// TIA Portal V17 export
// export: Created 2025-06-20T10:25:51.5107314Z, ExportSetting WithDefaults, DisplayName Totally Integrated Automation Portal, DisplayVersion V17 Update 8, DisplayName TIA Portal Openness, DisplayVersion V17 Update 8, DisplayName TIA Portal Version Control Interface, DisplayVersion V17, DisplayName SINAMICS Startdrive Advanced, DisplayVersion V17 SP2, DisplayName SINAMICS Startdrive G110M, G120, G120C, G120D, G120P, G115D, DisplayVersion V17 SP2, DisplayName SINAMICS Startdrive G130, G150, S120, S150, SINAMICS MV, S210, DisplayVersion V17 SP2, DisplayName STEP 7 Professional, DisplayVersion V17 Update 8, DisplayName SINUMERIK ONE STEP 7 Toolbox, DisplayVersion V17 Update 12, DisplayName SINUMERIK ONE PLC Basic Program Plus, DisplayVersion V17 Update 12, DisplayName SINUMERIK 840D sl STEP 7 Toolbox, DisplayVersion V17 Update 12, DisplayName STEP 7 Safety, DisplayVersion V17 Update 6, DisplayName WinCC Advanced, DisplayVersion V17 Update 8
DATA_BLOCK "DB450_ALARMS_WARNINGS_OPC_UA"   // DB450
{ S7_Optimized_Access := 'FALSE' }
VERSION : 0.1
// stored: AutoNumber false, DBAccessibleFromOPCUA true, DBAccessibleFromWebserver true, IsOnlyStoredInLoadMemory false, IsWriteProtectedInAS false
   VAR RETAIN
      ALARMS : Struct   // ALARMS MAIN NODE
         GENERAL : Struct   // GENERAL ALARMS
            "700008" : Bool;   // (RHP_SEOC) C11 Nreal<Nref
            "700009" : Bool;   // (RHP_SEOC) C11 ROTATION CONTROL FAULT
            "700010" : Bool;   // (RHP_SEOC) C11 COOLING SYSTEM OFF
            "700011" : Bool;   // (RHP_SEOC) C11 MQL OR COOLANT SYSTEM OFF
            "700012" : Bool;   // (SEOC) C11 HIGH TEMPERATURE ALARM
            "700013" : Bool;   // (SEOC) C11 PTC SENSOR HIGH TEMPERATURE ALARM
            "700014" : Bool;   // (SEOC) C11 VPM NOT READY ALARM
            "700016" : Bool;   // (RHP_SEOC) C12 Nreal<Nref
            "700017" : Bool;   // (RHP_SEOC) C12 ROTATION CONTROL FAULT
            "700018" : Bool;   // (RHP_SEOC) C12 COOLING SYSTEM OFF
            "700019" : Bool;   // (RHP_SEOC) C12 MQL OR COOLANT SYSTEM OFF
            "700020" : Bool;   // (SEOC) C12 HIGH TEMPERATURE ALARM
            "700021" : Bool;   // (SEOC) C12 PTC SENSOR HIGH TEMPERATURE ALARM
            "700022" : Bool;   // (SEOC) C12 VPM NOT READY ALARM
            "700024" : Bool;   // (RHP_SEOC) C13 Nreal<Nref
            "700025" : Bool;   // (RHP_SEOC) C13 ROTATION CONTROL FAULT
            "700026" : Bool;   // (RHP_SEOC) C13 COOLING SYSTEM OFF
            "700027" : Bool;   // (RHP_SEOC) C13 MQL OR COOLANT SYSTEM OFF
            "700028" : Bool;   // (SEOC) C13 HIGH TEMPERATURE ALARM
            "700029" : Bool;   // (SEOC) C13 PTC SENSOR HIGH TEMPERATURE ALARM
            "700030" : Bool;   // (SEOC) C13 VPM NOT READY ALARM
            "700032" : Bool;   // (RHP_SEOC) C14 Nreal<Nref
            "700033" : Bool;   // (RHP_SEOC) C14 ROTATION CONTROL FAULT
            "700034" : Bool;   // (RHP_SEOC) C14 COOLING SYSTEM OFF
            "700035" : Bool;   // (RHP_SEOC) C14 MQL OR COOLANT SYSTEM OFF
            "700036" : Bool;   // (SEOC) C14 HIGH TEMPERATURE ALARM
            "700037" : Bool;   // (SEOC) C14 PTC SENSOR HIGH TEMPERATURE ALARM
            "700038" : Bool;   // (SEOC) C14 VPM NOT READY ALARM
            "700056" : Bool;   // (RHP_SEOC) C21 Nreal<Nref
            "700057" : Bool;   // (RHP_SEOC) C21 ROTATION CONTROL FAULT
            "700058" : Bool;   // (RHP_SEOC) C21 COOLING SYSTEM OFF
            "700059" : Bool;   // (RHP_SEOC) C21 MQL OR COOLANT SYSTEM OFF
            "700060" : Bool;   // (SEOC) C21 HIGH TEMPERATURE ALARM
            "700061" : Bool;   // (SEOC) C21 PTC SENSOR HIGH TEMPERATURE ALARM
            "700062" : Bool;   // (SEOC) C21 VPM NOT READY ALARM
            "700072" : Bool;   // (RHP_SEOC) C23 Nreal<Nref
            "700073" : Bool;   // (RHP_SEOC) C23 ROTATION CONTROL FAULT
            "700074" : Bool;   // (RHP_SEOC) C23 COOLING SYSTEM OFF
            "700075" : Bool;   // (RHP_SEOC) C23 MQL OR COOLANT SYSTEM OFF
            "700076" : Bool;   // (SEOC) C23 HIGH TEMPERATURE ALARM
            "700077" : Bool;   // (SEOC) C23 PTC SENSOR HIGH TEMPERATURE ALARM
            "700078" : Bool;   // (SEOC) C23 VPM NOT READY ALARM
            "700080" : Bool;   // (RHP_SEOC) C24 Nreal<Nref
            "700081" : Bool;   // (RHP_SEOC) C24 ROTATION CONTROL FAULT
            "700082" : Bool;   // (RHP_SEOC) C24 COOLING SYSTEM OFF
            "700083" : Bool;   // (RHP_SEOC) C24 MQL OR COOLANT SYSTEM OFF
            "700084" : Bool;   // (SEOC) C24 HIGH TEMPERATURE ALARM
            "700085" : Bool;   // (SEOC) C24 PTC SENSOR HIGH TEMPERATURE ALARM
            "700086" : Bool;   // (SEOC) C24 VPM NOT READY ALARM
            "700104" : Bool;   // (IS_SEOC) AXIS E10 NOT REFERENCED
            "700111" : Bool;   // (IS_SEOC) AXIS X13 NOT REFERENCED
            "700113" : Bool;   // (IS_SEOC) AXIS Z13 NOT REFERENCED
            "700115" : Bool;   // (IS_SEOC) AXIS W11 NOT REFERENCED
            "700117" : Bool;   // (IS_SEOC) AXIS E20 NOT REFERENCED
            "700120" : Bool;   // (IS_SEOC) AXIS C22 NOT REFERENCED
            "700124" : Bool;   // (IS_SEOC) AXIS X23 NOT REFERENCED
            "700126" : Bool;   // (IS_SEOC) AXIS Z23 NOT REFERENCED
            "700128" : Bool;   // (IS_SEOC) AXIS W21 NOT REFERENCED
            "700133" : Bool;   // (IS_SEOC) AXIS C31 NOT REFERENCED
            "700400" : Bool;   // (IS) CHANNEL 1 NOT IN SOFT MODE. CHECK 20150[20]=2
            "700401" : Bool;   // (IS) PROGRAM SELECTION FAULT CHANNEL 1
            "700402" : Bool;   // (IS_SEOC) CHANNEL 1 READ AXES POSITION ALARM
            "700416" : Bool;   // (IS) CHANNEL 2 NOT IN SOFT MODE. CHECK 20150[20]=2
            "700417" : Bool;   // (IS) PROGRAM SELECTION FAULT CHANNEL 2
            "700418" : Bool;   // (IS_SEOC) CHANNEL 2 READ AXES POSITION ALARM
            "700432" : Bool;   // (IS) CHANNEL 3 NOT IN SOFT MODE. CHECK 20150[20]=2
            "700433" : Bool;   // (IS) PROGRAM SELECTION FAULT CHANNEL 3
            "700434" : Bool;   // (IS_SEOC) CHANNEL 3 READ AXES POSITION ALARM
            "700448" : Bool;   // (IS) CHANNEL 4 NOT IN SOFT MODE. CHECK 20150[20]=2
            "700449" : Bool;   // (IS) PROGRAM SELECTION FAULT CHANNEL 4
            "700450" : Bool;   // (IS_SEOC) CHANNEL 4 READ AXES POSITION ALARM
            "700464" : Bool;   // (IS) CHANNEL 5 NOT IN SOFT MODE. CHECK 20150[20]=2
            "700465" : Bool;   // (IS) PROGRAM SELECTION FAULT CHANNEL 5
            "700466" : Bool;   // (IS_SEOC) CHANNEL 5 READ AXES POSITION ALARM
            "700480" : Bool;   // (IS) CHANNEL 6 NOT IN SOFT MODE. CHECK 20150[20]=2
            "700481" : Bool;   // (IS) PROGRAM SELECTION FAULT CHANNEL 6
            "700482" : Bool;   // (IS_SEOC) CHANNEL 6 READ AXES POSITION ALARM
            "700496" : Bool;   // (IS) CHANNEL 7 NOT IN SOFT MODE. CHECK 20150[20]=2
            "700497" : Bool;   // (IS) PROGRAM SELECTION FAULT CHANNEL 7
            "700498" : Bool;   // (IS_SEOC) CHANNEL 7 READ AXES POSITION ALARM
            "700512" : Bool;   // (IS) CHANNEL 8 NOT IN SOFT MODE. CHECK 20150[20]=2
            "700513" : Bool;   // (IS) PROGRAM SELECTION FAULT CHANNEL 8
            "700514" : Bool;   // (IS_SEOC) CHANNEL 8 READ AXES POSITION ALARM
            "700528" : Bool;   // (IS) CHANNEL 9 NOT IN SOFT MODE. CHECK 20150[20]=2
            "700529" : Bool;   // (IS) PROGRAM SELECTION FAULT CHANNEL 9
            "700530" : Bool;   // (IS_SEOC) CHANNEL 9 READ AXES POSITION ALARM
            "700560" : Bool;   // (IS) FEEDBACK EMERGENCY STOP ALARM
            "700561" : Bool;   // (IS) FEEDBACK SAFETY DOORS UNIT 1 ALARM
            "700562" : Bool;   // (IS) FEEDBACK POWER ENABLE ALARM
            "700563" : Bool;   // (IS) FEEDBACK MACHINE TO ROBOT CELL SAFETY DOORS ALARM
            "700567" : Bool;   // (IS) FEEDBACK MACHINE EMERGENCY STOP ALARM
            "700568" : Bool;   // (IS) FEEDBACK LASER ENABLE CONDITIONS ALARM
            "700569" : Bool;   // (IS) FEEDBACK SAFETY DOORS UNIT 2 ALARM
            "700584" : Bool;   // (IS) TEST STOP SEQUENCE TIME EXCEEDED
            "700592" : Bool;   // (IS) BRAKE TEST AXIS X13 ALARM
            "700593" : Bool;   // (IS) BRAKE TEST AXIS W11 ALARM
            "700594" : Bool;   // (IS) BRAKE TEST AXIS Z13 ALARM
            "700595" : Bool;   // (IS) BRAKE TEST AXIS X23 ALARM
            "700596" : Bool;   // (IS) BRAKE TEST AXIS W21 ALARM
            "700597" : Bool;   // (IS) BRAKE TEST AXIS Z23 ALARM
            "700598" : Bool;   // (IS) BRAKE TEST AXIS C11 ALARM
            "700599" : Bool;   // (IS) BRAKE TEST AXIS C12 ALARM
            "700600" : Bool;   // (IS) BRAKE TEST AXIS C13 ALARM
            "700601" : Bool;   // (IS) BRAKE TEST AXIS C14 ALARM
            "700602" : Bool;   // (IS) BRAKE TEST AXIS C21 ALARM
            "700603" : Bool;   // (IS) BRAKE TEST AXIS C22 ALARM
            "700604" : Bool;   // (IS) BRAKE TEST AXIS C23 ALARM
            "700605" : Bool;   // (IS) BRAKE TEST AXIS C24 ALARM
            "700606" : Bool;   // (IS) BRAKE TEST AXIS C31 ALARM
            "700624" : Bool;   // (IS) TEST STOP INTERNAL PULSES ALARM AXIS E10
            "700625" : Bool;   // (IS) TEST STOP INTERNAL PULSES ALARM AXIS -
            "700626" : Bool;   // (IS) TEST STOP INTERNAL PULSES ALARM AXIS C11
            "700627" : Bool;   // (IS) TEST STOP INTERNAL PULSES ALARM AXIS C12
            "700632" : Bool;   // (IS) TEST STOP INTERNAL PULSES ALARM AXIS C13
            "700633" : Bool;   // (IS) TEST STOP INTERNAL PULSES ALARM AXIS C14
            "700634" : Bool;   // (IS) TEST STOP INTERNAL PULSES ALARM AXIS -
            "700635" : Bool;   // (IS) TEST STOP INTERNAL PULSES ALARM AXIS X13
            "700640" : Bool;   // (IS) TEST STOP INTERNAL PULSES ALARM AXIS -
            "700641" : Bool;   // (IS) TEST STOP INTERNAL PULSES ALARM AXIS W11
            "700642" : Bool;   // (IS) TEST STOP INTERNAL PULSES ALARM AXIS -
            "700643" : Bool;   // (IS) TEST STOP INTERNAL PULSES ALARM AXIS Z13
            "700644" : Bool;   // (IS) TEST STOP INTERNAL PULSES ALARM AXIS -
            "700645" : Bool;   // (IS) TEST STOP INTERNAL PULSES ALARM AXIS -
            "700646" : Bool;   // (IS) TEST STOP INTERNAL PULSES ALARM AXIS E20
            "700647" : Bool;   // (IS) TEST STOP INTERNAL PULSES ALARM AXIS -
            "700648" : Bool;   // (IS) TEST STOP INTERNAL PULSES ALARM AXIS C21
            "700649" : Bool;   // (IS) TEST STOP INTERNAL PULSES ALARM AXIS C22
            "700650" : Bool;   // (IS) TEST STOP INTERNAL PULSES ALARM AXIS C23
            "700651" : Bool;   // (IS) TEST STOP INTERNAL PULSES ALARM AXIS C24
            "700652" : Bool;   // (IS) TEST STOP INTERNAL PULSES ALARM AXIS -
            "700653" : Bool;   // (IS) TEST STOP INTERNAL PULSES ALARM AXIS X23
            "700654" : Bool;   // (IS) TEST STOP INTERNAL PULSES ALARM AXIS -
            "700655" : Bool;   // (IS) TEST STOP INTERNAL PULSES ALARM AXIS W21
            "700656" : Bool;   // (IS) TEST STOP INTERNAL PULSES ALARM AXIS -
            "700657" : Bool;   // (IS) TEST STOP INTERNAL PULSES ALARM AXIS Z23
            "700658" : Bool;   // (IS) TEST STOP INTERNAL PULSES ALARM AXIS -
            "700659" : Bool;   // (IS) TEST STOP INTERNAL PULSES ALARM AXIS -
            "700660" : Bool;   // (IS) TEST STOP INTERNAL PULSES ALARM AXIS C31
            "700661" : Bool;   // TEST STOP INTERNAL PULSES ALARM AXIS -
            "700662" : Bool;   // TEST STOP INTERNAL PULSES ALARM AXIS -
            "700700" : Bool;   // (IS) ERROR I-DEVICE SAFE SENDDP POWDER FEEDER ALARM
            "700701" : Bool;   // (IS) ERROR I-DEVICE SAFE SENDDP ROBOT CELL ALARM
            "700710" : Bool;   // (IS) ERROR I-DEVICE SAFE RCVDP POWDER FEEDER ALARM
            "700711" : Bool;   // (IS) ERROR I-DEVICE SAFE RCVDP ROBOT CELL ALARM
            "702400" : Bool;   // (IS) MACHINING SEQUENCE TIME EXCEEDED
            "702443" : Bool;   // (IS_SEOC) UNIT 1 STATION 3 CALIBRATION TIME EXCEEDED
            "702446" : Bool;   // (IS_SEOC) UNIT 1 STATION 0 PART CHECK TIME EXCEEDED
            "702448" : Bool;   // (IS_SEOC) PART CYCLE UNIT 1 SEQUENCE TIME EXCEEDED
            "702451" : Bool;   // (IS_SEOC) UNIT 1 STATION 0 SEQUENCE TIME EXCEEDED
            "702452" : Bool;   // (IS_SEOC) UNIT 1 STATION 1 SEQUENCE TIME EXCEEDED
            "702454" : Bool;   // (IS_SEOC) UNIT 1 STATION 3 SEQUENCE TIME EXCEEDED
            "702455" : Bool;   // (IS_SEOC) UNIT 1 STATION 4 SEQUENCE TIME EXCEEDED
            "702458" : Bool;   // (IS_SEOC) CLEAN FIXTURE UNIT 1 SEQUENCE TIME EXCEEDED
            "702459" : Bool;   // (IS_SEOC) GUIDEWAY CLEAN UNIT 1 SEQUENCE TIME EXCEEDED
            "702460" : Bool;   // (IS_SEOC) NOZZLE CLEAN UNIT 1 SEQUENCE TIME EXCEEDED
            "702461" : Bool;   // (IS_SEOC) MAINTENANCE UNIT 1 SEQUENCE TIME EXCEEDED
            "702462" : Bool;   // (IS_SEOC) RETURN TO HOME POSITION UNIT 1 STATION 0 SEQUENCE TIME EXCEEDED
            "702463" : Bool;   // (IS_SEOC) RETURN TO HOME POSITION UNIT 1 STATION 1 SEQUENCE TIME EXCEEDED
            "702465" : Bool;   // (IS_SEOC) RETURN TO HOME POSITION UNIT 1 STATION 3 SEQUENCE TIME EXCEEDED
            "702466" : Bool;   // (IS_SEOC) RETURN TO HOME POSITION UNIT 1 STATION 4 SEQUENCE TIME EXCEEDED
            "702468" : Bool;   // (IS_SEOC) UNIT 1 STATION 3 CAMERA LASER CALIBRATION SEQUENCE TIME EXCEEDED
            "702469" : Bool;   // (IS_SEOC) UNIT 1 STATION 3 CAMERA NOZZLE CALIBRATION SEQUENCE TIME EXCEEDED
            "702470" : Bool;   // (IS_SEOC) UNIT 1 STATION 3 CAMERA JET CALIBRATION SEQUENCE TIME EXCEEDED
            "702471" : Bool;   // (IS_SEOC) UNIT 1 STATION 3 CAMERA CLADDING CALIBRATION SEQUENCE TIME EXCEEDED
            "702482" : Bool;   // (IS_SEOC) UNIT 2 STATION 2 CALIBRATION TIME EXCEEDED
            "702483" : Bool;   // (IS_SEOC) UNIT 2 STATION 3 CALIBRATION TIME EXCEEDED
            "702486" : Bool;   // (IS_SEOC) UNIT 2 STATION 0 PART CHECK TIME EXCEEDED
            "702488" : Bool;   // (IS_SEOC) PART CYCLE UNIT 2 SEQUENCE TIME EXCEEDED
            "702491" : Bool;   // (IS_SEOC) UNIT 2 STATION 0 SEQUENCE TIME EXCEEDED
            "702492" : Bool;   // (IS_SEOC) UNIT 2 STATION 1 SEQUENCE TIME EXCEEDED
            "702493" : Bool;   // (IS_SEOC) UNIT 2 STATION 2 SEQUENCE TIME EXCEEDED
            "702494" : Bool;   // (IS_SEOC) UNIT 2 STATION 3 SEQUENCE TIME EXCEEDED
            "702495" : Bool;   // (IS_SEOC) UNIT 2 STATION 4 SEQUENCE TIME EXCEEDED
            "702498" : Bool;   // (IS_SEOC) CLEAN FIXTURE UNIT 2 SEQUENCE TIME EXCEEDED
            "702499" : Bool;   // (IS_SEOC) GUIDEWAY CLEAN UNIT 2 SEQUENCE TIME EXCEEDED
            "702500" : Bool;   // (IS_SEOC) NOZZLE CLEAN UNIT 2 SEQUENCE TIME EXCEEDED
            "702501" : Bool;   // (IS_SEOC) MAINTENANCE UNIT 2 SEQUENCE TIME EXCEEDED
            "702502" : Bool;   // (IS_SEOC) RETURN TO HOME POSITION UNIT 2 STATION 0 SEQUENCE TIME EXCEEDED
            "702503" : Bool;   // (IS_SEOC) RETURN TO HOME POSITION UNIT 2 STATION 1 SEQUENCE TIME EXCEEDED
            "702504" : Bool;   // (IS_SEOC) RETURN TO HOME POSITION UNIT 2 STATION 2 SEQUENCE TIME EXCEEDED
            "702505" : Bool;   // (IS_SEOC) RETURN TO HOME POSITION UNIT 2 STATION 3 SEQUENCE TIME EXCEEDED
            "702506" : Bool;   // (IS_SEOC) RETURN TO HOME POSITION UNIT 2 STATION 4 SEQUENCE TIME EXCEEDED
            "702508" : Bool;   // (IS_SEOC) UNIT 2 STATION 3 CAMERA LASER CALIBRATION SEQUENCE TIME EXCEEDED
            "702509" : Bool;   // (IS_SEOC) UNIT 2 STATION 3 CAMERA NOZZLE CALIBRATION SEQUENCE TIME EXCEEDED
            "702510" : Bool;   // (IS_SEOC) UNIT 2 STATION 3 CAMERA JET CALIBRATION SEQUENCE TIME EXCEEDED
            "702511" : Bool;   // (IS_SEOC) UNIT 2 STATION 3 CAMERA CLADDING CALIBRATION SEQUENCE TIME EXCEEDED
            "702515" : Bool;   // (IS_SEOC) UNIT 03 MEASURING STATION SEQUENCE TIME EXCEEDED
            "702516" : Bool;   // (IS_SEOC) UNIT 03 MEASURING STATION CALIBRATION SEQUENCE TIME EXCEEDED
            "702518" : Bool;   // (IS_SEOC) RETURN TO HOME POSITION UNIT 03 MEASURING SEQUENCE TIME EXCEEDED
            "702640" : Bool;   // (IS) ANY AXIS OR CHANNEL BYPASSED
            "702641" : Bool;   // (IS) ANY PROGRAMMING FAULT PRESENT
            "702642" : Bool;   // (IS) CHECK NETWORK LOGIC ALARM
            "702648" : Bool;   // (IS) LINE CONTACTOR FEEDBACK 1 ALARM
            "702649" : Bool;   // (IS) LINE CONTACTOR FEEDBACK 2 ALARM
            "702656" : Bool;   // (IS) INFEED MODULE 1 NOT READY ALARM
            "702657" : Bool;   // (SEOC) INFEED MODULE 1 OVERTEMPERATURE ALARM
            "702658" : Bool;   // (IS) INFEED MODULE 2 NOT READY ALARM
            "702659" : Bool;   // (SEOC) INFEED MODULE 2 OVERTEMPERATURE ALARM
            "702660" : Bool;   // (SEOC) NCU HEAT SINK TEMPERATURE ALARM
            "702661" : Bool;   // (SEOC) NCU LOW BATTERY ALARM
            "702662" : Bool;   // (SEOC) NCU AIR TEMPERATURE ALARM
            "702663" : Bool;   // (IS) NCK ALARM
            "702672" : Bool;   // (IS) ELECTRICAL CABINET MAIN SWITCH CIRCUIT BREAKER TRIPPED
            "702673" : Bool;   // (SEOC) ELECTRICAL CABINET COOLING UNIT 1 CIRCUIT BREAKER TRIPPED
            "702674" : Bool;   // (SEOC) ELECTRICAL CABINET COOLING UNIT 2 CIRCUIT BREAKER TRIPPED
            "702675" : Bool;   // (IS) CONTROL VOLTAGE ON ALARM
            "702677" : Bool;   // (IS) ELECTRICAL CABINET SINAMICS DRIVES CIRCUIT BREAKER 24VDC TRIPPED 1
            "702678" : Bool;   // (IS) ELECTRICAL CABINET SINAMICS DRIVES CIRCUIT BREAKER 24VDC TRIPPED 2
            "702681" : Bool;   // (IS) ELECTRICAL CABINET QFC03 CIRCUIT BREAKER TRIPPED
            "702682" : Bool;   // (IS) ELECTRICAL CABINET SINAMICS CIRCUIT BREAKER TRIPPED
            "702683" : Bool;   // (IS) FEEDBACK MAIN SWITCH OFF ALARM
            "702684" : Bool;   // (IS) ELECTRICAL CABINET OVERVOLTAGE
            "702686" : Bool;   // (SEOC) ELECTRICAL CABINET OVERTEMPERATURE ALARM
            "702689" : Bool;   // (SEOC) ELECTRICAL CABINET COOLING UNIT 1 ALARM
            "702690" : Bool;   // (SEOC) ELECTRICAL CABINET COOLING UNIT 2 ALARM
            "702694" : Bool;   // (SEOC) SENTRON PAC OVERVOLTAGE
            "702695" : Bool;   // (SEOC) SENTRON PAC OVERCURRENT
            "702697" : Bool;   // (SEOC) SENTRON PAC UNDERVOLTAGE
            "702700" : Bool;   // (IS) POWER SUPPLY DEVICE 1 ALARM
            "702703" : Bool;   // (IS) POWER SUPPLY 24V DEVICE 1 NOT OK ALARM
            "702704" : Bool;   // (IS) POWER SUPPLY 24V DEVICE 2 NOT OK ALARM
            "702705" : Bool;   // (IS) POWER SUPPLY 24V DEVICE 3 NOT OK ALARM
            "702706" : Bool;   // (IS) POWER SUPPLY 24V DEVICE 4 NOT OK ALARM
            "702707" : Bool;   // (IS) POWER SUPPLY 24V DEVICE 5 NOT OK ALARM
            "702708" : Bool;   // (IS) POWER SUPPLY 24V DEVICE 6 NOT OK ALARM
            "702709" : Bool;   // (IS) PILZ EMERGENCY STOP OK ALARM
            "702710" : Bool;   // (SEOC) SITOP BATTERY NOT OK ALARM
            "702711" : Bool;   // (SEOC) SITOP BATTERY ALARM
            "702714" : Bool;   // (IS) ETHERNET SWITCH 1 ALARM
            "702715" : Bool;   // (IS) ETHERNET SWITCH 2 ALARM
            "702716" : Bool;   // (IS) ETHERNET SWITCH 3 ALARM
            "702717" : Bool;   // (IS) ETHERNET SWITCH 4 ALARM
            "702718" : Bool;   // (IS) PROFINET CONTROL UNIT FAULT ALARM
            "702720" : Bool;   // (IS) ELECTRONIC CIRCUIT BREAKER 1 TRIPPED
            "702721" : Bool;   // (IS) ELECTRONIC CIRCUIT BREAKER 2 TRIPPED
            "702722" : Bool;   // (IS) ELECTRONIC CIRCUIT BREAKER 3 TRIPPED
            "702723" : Bool;   // (IS) ELECTRONIC CIRCUIT BREAKER 4 TRIPPED
            "702726" : Bool;   // (IS) FC40 CIRCUIT BREAKER TRIPPED
            "702727" : Bool;   // (IS) QB02 CIRCUIT BREAKER TRIPPED
            "702776" : Bool;   // (IS) SINAMICS CIRCUIT BREAKER TRIPPED ALARM
            "702777" : Bool;   // (IS) LASER UNIT 1 CIRCUIT BREAKER TRIPPED ALARM
            "702778" : Bool;   // (IS) LASER UNIT 2 CIRCUIT BREAKER TRIPPED ALARM
            "702779" : Bool;   // (IS) OERLIKON UNIT 1 CIRCUIT BREAKER TRIPPED ALARM
            "702780" : Bool;   // (IS) OERLIKON UNIT 2 CIRCUIT BREAKER TRIPPED ALARM
            "702781" : Bool;   // (IS) HEATER CIRCUIT BREAKER TRIPPED ALARM
            "702782" : Bool;   // (IS) CAMERAS CIRCUIT BREAKER 1 TRIPPED ALARM
            "702784" : Bool;   // (IS) STIRRER CIRCUIT BREAKER TRIPPED ALARM
            "702785" : Bool;   // (IS) COOLING CIRCUIT BREAKER TRIPPED ALARM
            "702786" : Bool;   // (IS) HOPPERS CIRCUIT BREAKER TRIPPED ALARM
            "702789" : Bool;   // (IS) ROBOT CELL COOLING CIRCUIT BREAKER TRIPPED ALARM
            "702790" : Bool;   // (SEOC) CIRCUIT BREAKER TRIPPED LIGHT STATION 3 ALARM
            "702793" : Bool;   // (IS) LASER UNIT 1 OK ALARM
            "702794" : Bool;   // (IS) LASER UNIT 2 OK ALARM
            "702795" : Bool;   // (SEOC) ROBOT CELL BREAKER ALARM
            "702800" : Bool;   // (IS) MAIN OPERATOR PANEL EMERGENCY STOP ACTIVE
            "702806" : Bool;   // (IS) HT10 EMERGENCY STOP ACTIVE
            "702809" : Bool;   // (IS) EMERGENCY STOP ACTIVE
            "702812" : Bool;   // (IS) ROBOT CELL EMERGENCY STOP ACTIVE
            "702814" : Bool;   // (IS) HT10 NOT READY ALARM
            "702815" : Bool;   // (IS) HT10 ERROR STATE ALARM
            "702820" : Bool;   // (SEOC) SAFETY BYPASS KEY ALARM
            "702880" : Bool;   // (IS) PROFINET NETWORK ALARM
            "702881" : Bool;   // (SEOC) PROFINET NETWORK ALARM
            "702882" : Bool;   // (RHP_SEOC) PROFINET NETWORK ALARM
            "704000" : Bool;   // (IS) UNIT 1 MAIN SAFETY DOOR NOT CLOSED AND LOCKED
            "704001" : Bool;   // (IS) UNIT 1 MAIN SAFETY DOOR NOT POSSIBLE TO UNLOCK DEPRESSURIZE PNEUMATIC DRIVE
            "704002" : Bool;   // (IS) UNIT 1 MAIN SAFETY DOOR NOT OPEN ALARM
            "704003" : Bool;   // (IS) UNIT 1 STATION 02 UNIT SAFETY DOOR NOT CLOSED AND LOCKED
            "704004" : Bool;   // (IS) UNIT 1 STATION 02 UNIT SAFETY DOOR NOT POSSIBLE TO UNLOCK DEPRESSURIZE PNEUMATIC DRIVE
            "704005" : Bool;   // (IS) UNIT 1 STATION 02 SAFETY DOOR NOT OPEN ALARM
            "704006" : Bool;   // (IS) UNIT 1 STATION 04 SAFETY DOOR NOT CLOSED AND LOCKED
            "704007" : Bool;   // (IS) UNIT 1 STATION 04 SAFETY DOOR NOT POSSIBLE TO UNLOCK DEPRESSURIZE PNEUMATIC DRIVE
            "704008" : Bool;   // (IS) UNIT 1 STATION 04 SAFETY DOOR NOT OPEN ALARM
            "704009" : Bool;   // (IS) UNIT 2 MAIN SAFETY DOOR NOT CLOSED AND LOCKED
            "704010" : Bool;   // (IS) UNIT 2 MAIN SAFETY DOOR NOT POSSIBLE TO UNLOCK DEPRESSURIZE PNEUMATIC DRIVE
            "704011" : Bool;   // (IS) UNIT 2 MAIN SAFETY DOOR NOT OPEN ALARM
            "704012" : Bool;   // (IS) UNIT 2 STATION 02 SAFETY DOOR NOT CLOSED AND LOCKED
            "704013" : Bool;   // (IS) UNIT 2 STATION 02 SAFETY DOOR NOT POSSIBLE TO UNLOCK DEPRESSURIZE PNEUMATIC DRIVE
            "704014" : Bool;   // (IS) UNIT 2 STATION 02 SAFETY DOOR NOT OPEN ALARM
            "704015" : Bool;   // (IS) UNIT 2 STATION 04 SAFETY DOOR NOT CLOSED AND LOCKED
            "704016" : Bool;   // (IS) UNIT 2 STATION 04 SAFETY DOOR NOT POSSIBLE TO UNLOCK DEPRESSURIZE PNEUMATIC DRIVE
            "704017" : Bool;   // (IS) UNIT 2 STATION 04 SAFETY DOOR NOT OPEN ALARM
            "704240" : Bool;   // (IS_SEOC) MACHINE-ROBOT CELL PART TYPE DISCORDANCY
            "704241" : Bool;   // (IS) NO PART TYPE SELECTED
            "704242" : Bool;   // (IS) MACHINE RECIPES SEQUENCE TIME EXCEEDED ALARM
            "704243" : Bool;   // (SEOC) TEST 24 HOURS DONE
            "704264" : Bool;   // (IS) ALL FIXTURES SOFTWARE DISABLED
            "704265" : Bool;   // (IS_SEOC) ALL FIXTURES UNIT 1 DISABLED
            "704266" : Bool;   // (IS_SEOC) ALL FIXTURES UNIT 2 DISABLED
            "704275" : Bool;   // (IS) UNIT 1 FIXTURE 1&4 DISABLED SOFTWARE/HARDWARE PART PRESENT ALARM
            "704276" : Bool;   // (IS) UNIT 1 FIXTURE 2&3 DISABLED SOFTWARE/HARDWARE PART PRESENT ALARM
            "704277" : Bool;   // (IS) UNIT 2 FIXTURE 1&4 DISABLED SOFTWARE/HARDWARE PART PRESENT ALARM
            "704278" : Bool;   // (IS) UNIT 2 FIXTURE 2&3 DISABLED SOFTWARE/HARDWARE PART PRESENT ALARM
            "704400" : Bool;   // (IS) ROBOT CELL INTERLOCK LIFE BIT ALARM
            "704401" : Bool;   // (IS) PRODUCTION DISCORDANCY, ALL MACHINE FIXTURES ENABLED AND ROBOT CELL COOLING DEGRADED CYCLE ACTIVE (MORE THAN 1 COOLING DISABLED)
            "704402" : Bool;   // (IS_SEOC) ROBOT FAULT ALARM UNIT 1
            "704403" : Bool;   // (IS_SEOC) ROBOT FAULT ALARM UNIT 2
            "704404" : Bool;   // (IS_SEOC) MEASURING STATION FAULT FROM CELL
            "704410" : Bool;   // (IS) POWDER INTERLOCK LIFE BIT ALARM
            "704800" : Bool;   // (RHP_SEOC) PART REJECTED AFTER INSPECTION ON DEMAND
            "704808" : Bool;   // (SEOC) PART REJECTED AFTER INSPECTION ON DEMAND
            "704832" : Bool;   // (RHP_SEOC) QUALITY PART REJECTED AFTER PART COUNT REACHED
            "704840" : Bool;   // (SEOC) QUALITY PART REJECTED AFTER PART COUNT REACHED
            "704864" : Bool;   // (RHP_SEOC) PART REJECTED AFTER PART TYPE CHANGE
            "704872" : Bool;   // (SEOC) PART REJECTED AFTER PART TYPE CHANGE
            "704896" : Bool;   // (RHP_SEOC) PART REJECTED AFTER FIRST CYCLE
            "704904" : Bool;   // (SEOC) PART REJECTED AFTER FIRST CYCLE
         END_STRUCT;
         SERVICES : Struct   // SERVICES ALARMS
            "708080" : Bool;   // (IS) PNEUMATIC BRANCH P1 PRESSURE NOT REACHED ALARM
            "708081" : Bool;   // (IS) PNEUMATIC BRANCH P1 PRESSURE SWITCH ALARM
            "708082" : Bool;   // (IS) PNEUMATIC BRANCH P1 PRESSURE MISSING ALARM
            "708083" : Bool;   // (IS) PNEUMATIC CONNECTION SENSOR 1 ALARM
            "708084" : Bool;   // (IS) PNEUMATIC CONNECTION SENSOR 2 ALARM
            "708085" : Bool;   // (SEOC) PNEUMATIC DRIVE UNBLOCK PRESSURE ALARM
            "708086" : Bool;   // (SEOC) PNEUMATIC DRIVE PRESSURE UNBLOCK SWITCH ALARM
            "708087" : Bool;   // (SEOC) PNEUMATIC PRESSURIZATION ALARM
            "708088" : Bool;   // (SEOC) PNEUMATIC PRESSURIZATION SWITCH ALARM
            "708089" : Bool;   // (SEOC) PNEUMATIC UNIT 1 GRIPPER AIR PRESSURE ALARM
            "708090" : Bool;   // (SEOC) PNEUMATIC UNIT 1 GRIPPER AIR PRESSURE SWITCH ALARM
            "708091" : Bool;   // (SEOC) PNEUMATIC UNIT 1 LABERINT PRESSURE ALARM
            "708092" : Bool;   // (SEOC) PNEUMATIC UNIT 1 LABERINT PRESSURE SWITCH ALARM
            "708093" : Bool;   // (SEOC) PNEUMATIC UNIT 1 UPPER TABLE PRESSURE ALARM
            "708094" : Bool;   // (SEOC) PNEUMATIC UNIT 1 UPPER TABLE PRESSURE SWITCH ALARM
            "708095" : Bool;   // (SEOC) PNEUMATIC UNIT 1 LOWER TABLE PRESSURE ALARM
            "708096" : Bool;   // (SEOC) PNEUMATIC UNIT 1 LOWER TABLE PRESSURE SWITCH ALARM
            "708097" : Bool;   // (SEOC) PNEUMATIC UNIT 1 CART AXIS X PRESSURE ALARM
            "708098" : Bool;   // (SEOC) PNEUMATIC UNIT 1 CART AXIS X PRESSURE SWITCH ALARM
            "708099" : Bool;   // (SEOC) PNEUMATIC UNIT 1 STATION 3 MEASUREMENT UNIT PRESSURE ALARM
            "708100" : Bool;   // (SEOC) PNEUMATIC UNIT 1 STATION 3 MEASUREMENT UNIT PRESSURE SWITCH ALARM
            "708108" : Bool;   // (IS) PNEUMATIC INPUT FLOW ALARM
            "708109" : Bool;   // (IS) PNEUMATIC INPUT TEMPERATURE ALARM
            "708112" : Bool;   // (SEOC) PNEUMATIC UNIT 2 GRIPPER AIR PRESSURE ALARM
            "708113" : Bool;   // (SEOC) PNEUMATIC UNIT 2 GRIPPER AIR PRESSURE SWITCH ALARM
            "708114" : Bool;   // (SEOC) PNEUMATIC UNIT 2 LABERINT PRESSURE ALARM
            "708115" : Bool;   // (SEOC) PNEUMATIC UNIT 2 LABERINT PRESSURE SWITCH ALARM
            "708116" : Bool;   // (SEOC) PNEUMATIC UNIT 2 UPPER TABLE PRESSURE ALARM
            "708117" : Bool;   // (SEOC) PNEUMATIC UNIT 2 UPPER TABLE PRESSURE SWITCH ALARM
            "708118" : Bool;   // (SEOC) PNEUMATIC UNIT 2 LOWER TABLE PRESSURE ALARM
            "708119" : Bool;   // (SEOC) PNEUMATIC UNIT 2 LOWER TABLE PRESSURE SWITCH ALARM
            "708120" : Bool;   // (SEOC) PNEUMATIC UNIT 2 CART AXIS X PRESSURE ALARM
            "708121" : Bool;   // (SEOC) PNEUMATIC UNIT 2 CART AXIS X PRESSURE SWITCH ALARM
            "708122" : Bool;   // (SEOC) PNEUMATIC UNIT 2 STATION 3 MEASUREMENT UNIT PRESSURE ALARM
            "708123" : Bool;   // (SEOC) PNEUMATIC UNIT 2 STATION 3 MEASUREMENT UNIT PRESSURE SWITCH ALARM
            "708160" : Bool;   // (IS) GENERAL GAS SYSTEM PRESSURE ALARM
            "708400" : Bool;   // (IS_SEOC) MACHINE COOLING SYSTEM INPUT SENSOR FLOW LOW ALARM
            "708401" : Bool;   // (IS_SEOC) MACHINE COOLING SYSTEM INPUT SENSOR FLOW HIGH ALARM
            "708402" : Bool;   // (IS_SEOC) MACHINE COOLING SYSTEM INPUT SENSOR FLOW SETPOINT ALARM
            "708403" : Bool;   // (IS_SEOC) MACHINE COOLING SYSTEM INPUT SENSOR TEMPERATURE LOW ALARM
            "708404" : Bool;   // (IS_SEOC) MACHINE COOLING SYSTEM INPUT SENSOR TEMPERATURE HIGH ALARM
            "708405" : Bool;   // (IS_SEOC) MACHINE COOLING SYSTEM INPUT SENSOR TEMPERATURE SETPOINT ALARM
            "708407" : Bool;   // (IS_SEOC) MACHINE COOLING SYSTEM OUTPUT SENSOR FLOW LOW ALARM
            "708408" : Bool;   // (IS_SEOC) MACHINE COOLING SYSTEM OUTPUT SENSOR FLOW HIGH ALARM
            "708409" : Bool;   // (IS_SEOC) MACHINE COOLING SYSTEM OUTPUT SENSOR FLOW SETPOINT ALARM
            "708410" : Bool;   // (IS_SEOC) MACHINE COOLING SYSTEM OUTPUT SENSOR TEMPERATURE LOW ALARM
            "708411" : Bool;   // (IS_SEOC) MACHINE COOLING SYSTEM OUTPUT SENSOR TEMPERATURE HIGH ALARM
            "708412" : Bool;   // (IS_SEOC) MACHINE COOLING SYSTEM OUTPUT SENSOR TEMPERATURE SETPOINT ALARM
            "708417" : Bool;   // (SEOC) SHIELD AUXILIARY COOLING SYSTEM BREAKER TRIPPED ALARM
            "708418" : Bool;   // (SEOC) SHIELD AUXILIARY COOLING SYSTEM CONTACTOR FEEDBACK ALARM
            "708419" : Bool;   // (SEOC) SHIELD AUXILIARY COOLING SYSTEM LOW LEVEL ALARM
            "708420" : Bool;   // (SEOC) SHIELD AUXILIARY COOLING SYSTEM OVERTEMPERATURE ALARM
            "708423" : Bool;   // (SEOC) U01 SHIELD AUXILIARY COOLING SYSTEM FLOW FEEDBACK ALARM
            "708424" : Bool;   // (SEOC) U01 SHIELD AUXILIARY COOLING SYSTEM FLOW LOW ALARM
            "708425" : Bool;   // (SEOC) U01 SHIELD AUXILIARY COOLING SYSTEM FLOW HIGH ALARM
            "708426" : Bool;   // (SEOC) U01 SHIELD AUXILIARY COOLING SYSTEM TEMPERATURE LOW ALARM
            "708427" : Bool;   // (SEOC) U01 SHIELD AUXILIARY COOLING SYSTEM TEMPERATURE HIGH ALARM
            "708428" : Bool;   // (SEOC) U01 SHIELD AUXILIARY COOLING SYSTEM FLOW SETPOINT ALARM
            "708429" : Bool;   // (SEOC) U01 SHIELD AUXILIARY COOLING SYSTEM TEMPERATURE SETPOINT ALARM
            "708432" : Bool;   // (SEOC) U02 SHIELD AUXILIARY COOLING SYSTEM FLOW FEEDBACK ALARM
            "708433" : Bool;   // (SEOC) U02 SHIELD AUXILIARY COOLING SYSTEM FLOW LOW ALARM
            "708434" : Bool;   // (SEOC) U02 SHIELD AUXILIARY COOLING SYSTEM FLOW HIGH ALARM
            "708435" : Bool;   // (SEOC) U02 SHIELD AUXILIARY COOLING SYSTEM TEMPERATURE LOW ALARM
            "708436" : Bool;   // (SEOC) U02 SHIELD AUXILIARY COOLING SYSTEM TEMPERATURE HIGH ALARM
            "708437" : Bool;   // (SEOC) U02 SHIELD AUXILIARY COOLING SYSTEM FLOW SETPOINT ALARM
            "708438" : Bool;   // (SEOC) U02 SHIELD AUXILIARY COOLING SYTEM TEMPERATURE SETPOINT ALARM
            "708443" : Bool;   // (SEOC) COOLING BUFFER AUXILIARY COOLING SYSTEM BREAKER TRIPPED ALARM
            "708444" : Bool;   // (SEOC) COOLING BUFFER AUXILIARY COOLING SYSTEM CONTACTOR FEEDBACK ALARM
            "708445" : Bool;   // (SEOC) COOLING BUFFER AUXILIARY COOLING SYSTEM LOW LEVEL ALARM
            "708446" : Bool;   // (SEOC) COOLING BUFFER AUXILIARY COOLING SYSTEM OVERTEMPERATURE ALARM
            "708449" : Bool;   // (SEOC) U01 COOLING BUFFER AUXILIARY COOLING SYSTEM FLOW FEEDBACK ALARM
            "708450" : Bool;   // (SEOC) U01 COOLING BUFFER AUXILIARY COOLING SYSTEM FLOW LOW ALARM
            "708451" : Bool;   // (SEOC) U01 COOLING BUFFER AUXILIARY COOLING SYSTEM FLOW HIGH ALARM
            "708452" : Bool;   // (SEOC) U01 COOLING BUFFER AUXILIARY COOLING SYSTEM TEMPERATURE LOW ALARM
            "708453" : Bool;   // (SEOC) U01 COOLING BUFFER AUXILIARY COOLING SYSTEM TEMPERATURE HIGH ALARM
            "708454" : Bool;   // (SEOC) U01 COOLING BUFFER AUXILIARY COOLING SYSTEM FLOW SETPOINT ALARM
            "708455" : Bool;   // (SEOC) U01 COOLING BUFFER AUXILIARY COOLING SYSTEM TEMPERATURE SETPOINT ALARM
            "708458" : Bool;   // (SEOC) U02 COOLING BUFFER AUXILIARY COOLING SYSTEM FLOW FEEDBACK ALARM
            "708459" : Bool;   // (SEOC) U02 COOLING BUFFER AUXILIARY COOLING SYSTEM FLOW LOW ALARM
            "708460" : Bool;   // (SEOC) U02 COOLING BUFFER AUXILIARY COOLING SYSTEM FLOW HIGH ALARM
            "708461" : Bool;   // (SEOC) U02 COOLING BUFFER AUXILIARY COOLING SYSTEM TEMPERATURE LOW ALARM
            "708462" : Bool;   // (SEOC) U02 COOLING BUFFER AUXILIARY COOLING SYSTEM TEMPERATURE HIGH ALARM
            "708463" : Bool;   // (SEOC) U02 COOLING BUFFER AUXILIARY COOLING SYSTEM FLOW SETPOINT ALARM
            "708464" : Bool;   // (SEOC) U02 COOLING BUFFER AUXILIARY COOLING SYSTEM TEMPERATURE SETPOINT ALARM
            "708800" : Bool;   // (SEOC) PROGRESSIVE LUBRICATION CIRCUIT BREAKER TRIPPED
            "708801" : Bool;   // (SEOC) PROGRESSIVE LUBRICATION LOW LEVEL ALARM
            "708802" : Bool;   // (SEOC) PROGRESSIVE LUBRICATION OVERPRESSURE ALARM
            "708803" : Bool;   // (SEOC) PROGRESSIVE LUBRICATION BRANCH 1 CYCLE NOT DONE ALARM
            "708804" : Bool;   // (SEOC) PROGRESSIVE LUBRICATION BRANCH 2 CYCLE NOT DONE ALARM
            "708805" : Bool;   // (SEOC) PROGRESSIVE LUBRICATION BRANCH 3 CYCLE NOT DONE ALARM
            "708806" : Bool;   // (SEOC) PROGRESSIVE LUBRICATION BRANCH 4 CYCLE NOT DONE ALARM
            "708960" : Bool;   // (SEOC) MACHINE ASPIRATION SYSTEM ALARM
            "709040" : Bool;   // (IS_SEOC) UNIT 1 ASPIRATION SYSTEM PRESSURE TOO HIGH ALARM
            "709041" : Bool;   // (IS_SEOC) UNIT 1 ASPIRATION SYSTEM PRESSURE TOO LOW ALARM
            "709051" : Bool;   // (IS_SEOC) UNIT 1 STATION 1 ASPIRATION ACTIVATION SIMULTANEITY ALARM
            "709052" : Bool;   // (IS_SEOC) UNIT 1 STATION 1 ASPIRATION ACTIVATION TIME EXCEEDED ALARM
            "709053" : Bool;   // (IS_SEOC) UNIT 1 STATION 1 ASPIRATION ACTIVATION SWITCH ON ALARM
            "709054" : Bool;   // (IS_SEOC) UNIT 1 STATION 1 ASPIRATION ACTIVATION SWITCH OFF ALARM
            "709071" : Bool;   // (IS_SEOC) UNIT 1 STATION 3 ASPIRATION ACTIVATION SIMULTANEITY ALARM
            "709072" : Bool;   // (IS_SEOC) UNIT 1 STATION 3 ASPIRATION ACTIVATION TIME EXCEEDED ALARM
            "709073" : Bool;   // (IS_SEOC) UNIT 1 STATION 3 ASPIRATION ACTIVATION SWITCH ON ALARM
            "709074" : Bool;   // (IS_SEOC) UNIT 1 STATION 3 ASPIRATION ACTIVATION SWITCH OFF ALARM
            "709120" : Bool;   // (IS_SEOC) UNIT 2 ASPIRATION SYSTEM PRESSURE TOO HIGH ALARM
            "709121" : Bool;   // (IS_SEOC) UNIT 2 ASPIRATION SYSTEM PRESSURE TOO LOW ALARM
            "709131" : Bool;   // (IS_SEOC) UNIT 2 STATION 1 ASPIRATION ACTIVATION SIMULTANEITY ALARM
            "709132" : Bool;   // (IS_SEOC) UNIT 2 STATION 1 ASPIRATION ACTIVATION TIME EXCEEDED ALARM
            "709133" : Bool;   // (IS_SEOC) UNIT 2 STATION 1 ASPIRATION ACTIVATION SWITCH ON ALARM
            "709134" : Bool;   // (IS_SEOC) UNIT 2 STATION 1 ASPIRATION ACTIVATION SWITCH OFF ALARM
            "709151" : Bool;   // (IS_SEOC) UNIT 2 STATION 3 ASPIRATION ACTIVATION SIMULTANEITY ALARM
            "709152" : Bool;   // (IS_SEOC) UNIT 2 STATION 3 ASPIRATION ACTIVATION TIME EXCEEDED ALARM
            "709153" : Bool;   // (IS_SEOC) UNIT 2 STATION 3 ASPIRATION ACTIVATION SWITCH ON ALARM
            "709154" : Bool;   // (IS_SEOC) UNIT 2 STATION 3 ASPIRATION ACTIVATION SWITCH OFF ALARM
            "709161" : Bool;   // (IS_SEOC) UNIT 2 STATION 4 ASPIRATION ACTIVATION SIMULTANEITY ALARM
         END_STRUCT;
         UNIT_01 : Struct   // UNIT 01 ALARMS
            "716000" : Bool;   // (IS_SEOC) UNIT 1 FIXTURE 1 PART TYPE DISCORDANCY ALARM
            "716001" : Bool;   // (IS_SEOC) UNIT 1 FIXTURE 2 PART TYPE DISCORDANCY ALARM
            "716002" : Bool;   // (IS_SEOC) UNIT 1 FIXTURE 3 PART TYPE DISCORDANCY ALARM
            "716003" : Bool;   // (IS_SEOC) UNIT 1 FIXTURE 4 PART TYPE DISCORDANCY ALARM
            "716008" : Bool;   // (RHP_SEOC) UNIT 1 FIXTURE 1 PART PRESENT DISCORDANCY ALARM
            "716009" : Bool;   // (RHP_SEOC) UNIT 1 FIXTURE 2 PART PRESENT DISCORDANCY ALARM
            "716010" : Bool;   // (RHP_SEOC) UNIT 1 FIXTURE 3 PART PRESENT DISCORDANCY ALARM
            "716011" : Bool;   // (RHP_SEOC) UNIT 1 FIXTURE 4 PART PRESENT DISCORDANCY ALARM
            "716024" : Bool;   // (IS_SEOC) UNIT 1 FIXTURE 1 PART ORIENTATION DISCORDANCY ALARM
            "716025" : Bool;   // (IS_SEOC) UNIT 1 FIXTURE 2 PART ORIENTATION DISCORDANCY ALARM
            "716026" : Bool;   // (IS_SEOC) UNIT 1 FIXTURE 3 PART ORIENTATION DISCORDANCY ALARM
            "716027" : Bool;   // (IS_SEOC) UNIT 1 FIXTURE 4 PART ORIENTATION DISCORDANCY ALARM
            "716032" : Bool;   // (RHP_SEOC) UNIT 1 FIXTURE 1 NOT CLAMPED DURING MACHINING ALARM
            "716033" : Bool;   // (RHP_SEOC) UNIT 1 FIXTURE 2 NOT CLAMPED DURING MACHINING ALARM
            "716034" : Bool;   // (RHP_SEOC) UNIT 1 FIXTURE 3 NOT CLAMPED DURING MACHINING ALARM
            "716035" : Bool;   // (RHP_SEOC) UNIT 1 FIXTURE 4 NOT CLAMPED DURING MACHINING ALARM
            STATION_3_MEASURING : Struct   // STATION 3 MEASURING ALARMS
               "716480" : Bool;   // (IS_SEOC) UNIT 1 STATION 3 MEASURING LAST CALIBRATION OUT OF RANGE IN FIXTURE 1 ALARM
               "716481" : Bool;   // (IS_SEOC) UNIT 1 STATION 3 MEASURING LAST CALIBRATION OUT OF RANGE IN FIXTURE 2 ALARM
               "716482" : Bool;   // (IS_SEOC) UNIT 1 STATION 3 MEASURING LAST CALIBRATION OUT OF RANGE IN FIXTURE 3 ALARM
               "716483" : Bool;   // (IS_SEOC) UNIT 1 STATION 3 MEASURING LAST CALIBRATION OUT OF RANGE IN FIXTURE 4 ALARM
               "716488" : Bool;   // (IS_SEOC) UNIT 1 STATION 3 MEASURING COMPUTER CONNECTION CALL ERROR
               "716489" : Bool;   // (IS_SEOC) UNIT 1 STATION 3 MEASURING COMPUTER GET INDEX LIST CALL ERROR
               "716490" : Bool;   // (IS_SEOC) UNIT 1 STATION 3 MEASURING COMPUTER GET HANDLE LIST CALL ERROR
               "716491" : Bool;   // (IS_SEOC) UNIT 1 STATION 3 MEASURING COMPUTER GET METHOD LIST CALL ERROR
               "716492" : Bool;   // (IS_SEOC) UNIT 1 STATION 3 MEASURING COMPUTER RELEASE HANDLE LIST CALL ERROR
               "716493" : Bool;   // (IS_SEOC) UNIT 1 STATION 3 MEASURING COMPUTER RELEASE METHOD HANDLE LIST CALL ERROR
               "716494" : Bool;   // (IS_SEOC) UNIT 1 STATION 3 MEASURING COMPUTER DISCONNECT CALL ERROR
               "716500" : Bool;   // (IS_SEOC) UNIT 1 STATION 3 MEASURING COMPUTER ERROR: PROFILER CONFIGURATION (ISSUES WITH THE PROFILOMETER CONFIGURATION)
               "716501" : Bool;   // (IS_SEOC) UNIT 1 STATION 3 MEASURING COMPUTER ERROR: ANALYZER CONFIGURATION (ERROR OCCURRED WHILE VERIFYING THE CONFIGURATION FILES)
               "716502" : Bool;   // (IS_SEOC) UNIT 1 STATION 3 MEASURING COMPUTER ERROR: DMC STRUCTURE (PROBLEMS READING THE DMC STRING)
               "716503" : Bool;   // (IS_SEOC) UNIT 1 STATION 3 MEASURING COMPUTER ERROR: ACQUISITION (UNABLE TO ACQUIRE PROFILES FROM THE PROFILOMETER)
               "716504" : Bool;   // (IS_SEOC) UNIT 1 STATION 3 MEASURING COMPUTER ERROR: PROFILE INITIALIZATION (FAILED TO INITIALIZE THE PROFILOMETER)
               "716505" : Bool;   // (IS_SEOC) UNIT 1 STATION 3 MEASURING COMPUTER ERROR: DISTANCE CALCULATION (ISSUES EXECUTING THE DISTANCE CALCULATION ALGORITHM)
               "716506" : Bool;   // (IS_SEOC) UNIT 1 STATION 3 MEASURING COMPUTER ERROR: LAYER GROWTH ANALYSIS (ISSUES EXECUTING THE LAYER GROWTH ALGORITHM)
               "716507" : Bool;   // (IS_SEOC) UNIT 1 STATION 3 MEASURING COMPUTER ERROR: STORAGE ERROR (ERROR ATTEMPTING TO STORE DATA)
               "716508" : Bool;   // (IS_SEOC) UNIT 1 STATION 3 MEASURING COMPUTER ERROR: DATABASE CONNECTION ALARM (CALIBRATION CHECK OR MEASURE SAVE NOT POSSIBLE)
               "716509" : Bool;   // (IS_SEOC) UNIT 1 STATION 3 MEASURING COMPUTER ERROR: CALIBRATION PROCEDURE (CALIBRATION FAILED)
               "716510" : Bool;   // (IS_SEOC) UNIT 1 STATION 3 MEASURING COMPUTER ERROR: CALIBRATION MISSING IN FIXTURE 1 (CALIBRATION MISSING OR FILE NOT FOUND)
               "716511" : Bool;   // (IS_SEOC) UNIT 1 STATION 3 MEASURING COMPUTER ERROR: CALIBRATION MISSING IN FIXTURE 2 (CALIBRATION MISSING OR FILE NOT FOUND)
               "716512" : Bool;   // (IS_SEOC) UNIT 1 STATION 3 MEASURING COMPUTER ERROR: CALIBRATION MISSING IN FIXTURE 3 (CALIBRATION MISSING OR FILE NOT FOUND)
               "716513" : Bool;   // (IS_SEOC) UNIT 1 STATION 3 MEASURING COMPUTER ERROR: CALIBRATION MISSING IN FIXTURE 4 (CALIBRATION MISSING OR FILE NOT FOUND)
               "716514" : Bool;   // (IS_SEOC) UNIT 1 STATION 3 MEASURING COMPUTER ERROR: PLC-PC MAJOR VERSIONS MISMATCH
               "716515" : Bool;   // (SEOC) UNIT 1 STATION 3 MEASURING COMPUTER ERROR: INITIALIZING PROFILOMETER
               "716520" : Bool;   // (IS_SEOC) UNIT 1 STATION 3 MEASURING COMPUTER NOZZLE SURFACE DISTANCE UPDATE ALARM
               "716530" : Bool;   // (IS_SEOC) UNIT 1 STATION 3 MEASURING COMPUTER START NOOZLE MEASUREMENT METHOD CALL EXECUTION ERROR
               "716531" : Bool;   // (IS_SEOC) UNIT 1 STATION 3 MEASURING COMPUTER START NOOZLE MEASUREMENT METHOD WORKING OR BLOCKED ERROR
               "716546" : Bool;   // (IS_SEOC) UNIT 1 STATION 3 MEASURING COMPUTER START LAYER THICKNESS MEASUREMENT METHOD CALL EXECUTION ERROR
               "716547" : Bool;   // (IS_SEOC) UNIT 1 STATION 3 MEASURING COMPUTER START LAYER THICKNESS MEASUREMENT METHOD WORKING OR BLOCKED ERROR
               "716554" : Bool;   // (IS_SEOC) UNIT 1 STATION 3 MEASURING COMPUTER STOP LAYER THICKNESS MEASUREMENT METHOD CALL EXECUTION ERROR
               "716555" : Bool;   // (IS_SEOC) UNIT 1 STATION 3 MEASURING COMPUTER STOP LAYER THICKNESS MEASUREMENT METHOD WORKING OR BLOCKED ERROR
               "716562" : Bool;   // (IS_SEOC) UNIT 1 STATION 3 MEASURING COMPUTER CALIBRATING METHOD CALL EXECUTION ERROR
               "716563" : Bool;   // (IS_SEOC) UNIT 1 STATION 3 MEASURING COMPUTER CALIBRATING METHOD WORKING OR BLOCKED ERROR
               "716570" : Bool;   // (IS_SEOC) UNIT 1 STATION 3 MEASURING COMPUTER RESET METHOD CALL EXECUTION ERROR
               "716571" : Bool;   // (IS_SEOC) UNIT 1 STATION 3 MEASURING COMPUTER RESET METHOD WORKING OR BLOCKED ERROR
               "716578" : Bool;   // (IS_SEOC) UNIT 1 STATION 3 MEASURING COMPUTER READ VARIABLES METHOD CALL EXECUTION ERROR
               "716579" : Bool;   // (IS_SEOC) UNIT 1 STATION 3 MEASURING COMPUTER READ VARIABLES METHOD WORKING OR BLOCKED ERROR
            END_STRUCT;
            STATION_3_COAXIAL : Struct   // STATION 3 COAXIAL ALARMS
               "716640" : Bool;   // (IS_SEOC) UNIT 1 STATION 3 CAMERA COMPUTER ERROR: FAILED TO CONNECT TO CAMERA (UNABLE TO GET IMAGES FROM CAMERA)
               "716641" : Bool;   // (IS_SEOC) UNIT 1 STATION 3 CAMERA COMPUTER ERROR: FAILED TO SET CAMERA PARAMETERS (UNABLE TO SET CAMERA PARAMETERS (EXPOSURE-TIME & GAIN) FROM CURRENT IMAGES)
               "716642" : Bool;   // (IS_SEOC) UNIT 1 STATION 3 CAMERA COMPUTER ERROR: NEW LASER CALIBRATION REQUIRED (CURRENT CALIBRATION PARAMETERS DO NOT MEEST RECENT ANALYSIS REQUISITES)
               "716643" : Bool;   // (IS_SEOC) UNIT 1 STATION 3 CAMERA COMPUTER ERROR: NEW NOZZLE CALIBRATION REQUIRED (CURRENT CALIBRATION PARAMETERS DO NOT MEEST RECENT ANALYSIS REQUISITES)
               "716644" : Bool;   // (IS_SEOC) UNIT 1 STATION 3 CAMERA COMPUTER ERROR: NEW JET CALIBRATION REQUIRED (CURRENT CALIBRATION PARAMETERS DO NOT MEEST RECENT ANALYSIS REQUISITES)
               "716645" : Bool;   // (IS_SEOC) UNIT 1 STATION 3 CAMERA COMPUTER ERROR: NEW CLADDING CALIBRATION REQUIRED (CURRENT CALIBRATION PARAMETERS DO NOT MEEST RECENT ANALYSIS REQUISITES)
               "716646" : Bool;   // (IS_SEOC) UNIT 1 STATION 3 CAMERA COMPUTER ERROR: HIGH NUMBER OF DEAD PIXELS (THE NUMBER OF DEAD-PIXELS EXCEEDS A CONFIGURED NUMBER)
               "716647" : Bool;   // (IS_SEOC) UNIT 1 STATION 3 CAMERA COMPUTER ERROR: NO LIGHT DETECTED (NO LIGHT OR BLANK IMAGE DETECTED)
               "716648" : Bool;   // (IS_SEOC) UNIT 1 STATION 3 CAMERA COMPUTER ERROR: NO LASER DETECTED (NO LASER SPOT DETECTED)
               "716649" : Bool;   // (IS_SEOC) UNIT 1 STATION 3 CAMERA COMPUTER ERROR: NO NOZZLE DETECTED (UNABLE TO DETECT ANY CAPSULE-SHAPED NOZZLE IN THE IMAGE)
               "716651" : Bool;   // (IS_SEOC) UNIT 1 STATION 3 CAMERA COMPUTER ERROR: NO LASER PATTERN DETECTED (NO LASER PATERN HAS BEEN DETECTED IN THE IMAGE)
               "716652" : Bool;   // (IS_SEOC) UNIT 1 STATION 3 CAMERA COMPUTER ERROR: NOT ANALYZED
               "716653" : Bool;   // (IS_SEOC) UNIT 1 STATION 3 CAMERA COMPUTER ERROR: FAILED TO OBTAIN SCALE FACTOR
               "716654" : Bool;   // (IS_SEOC) UNIT 1 STATION 3 CAMERA COMPUTER ERROR: UNALIGNED POWDER FLOW VORTEX
               "716655" : Bool;   // (IS_SEOC) UNIT 1 STATION 3 CAMERA COMPUTER ERROR: JET MALFUNCTION
               "716656" : Bool;   // (IS_SEOC) UNIT 1 STATION 3 CAMERA COMPUTER ERROR: UNCALIBRATED
               "716657" : Bool;   // (IS_SEOC) UNIT 1 STATION 3 CAMERA COMPUTER ERROR: PLC-PC MAJOR VERSIONS MISMATCH
               "716658" : Bool;   // (IS_SEOC) UNIT 1 STATION 3 CAMERA COMPUTER ERROR: NO MELT POOL DETECTED
               "716659" : Bool;   // (IS_SEOC) UNIT 1 STATION 3 CAMERA COMPUTER ERROR: NO DATA BASE CONNECTION
               "716660" : Bool;   // (IS_SEOC) UNIT 1 STATION 3 CAMERA COMPUTER ERROR: NO HALO DETECTED
               "716661" : Bool;   // (IS_SEOC) UNIT 1 STATION 3 CAMERA COMPUTER ERROR: STORAGE ERROR
               "716662" : Bool;   // (SEOC) UNIT 1 STATION 3 CAMERA COMPUTER ERROR: INITIALIZING CAMERA
               "716663" : Bool;   // (IS_SEOC) UNIT 1 STATION 3 CAMERA COMPUTER ERROR: NOZZLE CONTAMINATION DETECTED
               "716664" : Bool;   // (IS_SEOC) UNIT 1 STATION 3 CAMERA COMPUTER ERROR: INVALID CONFIGURATION
               "716672" : Bool;   // (IS_SEOC) UNIT 1 STATION 3 CAMERA COMPUTER CONNECTION CALL ERROR
               "716673" : Bool;   // (IS_SEOC) UNIT 1 STATION 3 CAMERA COMPUTER GET INDEX LIST CALL ERROR
               "716674" : Bool;   // (IS_SEOC) UNIT 1 STATION 3 CAMERA COMPUTER GET HANDLE LIST CALL ERROR
               "716675" : Bool;   // (IS_SEOC) UNIT 1 STATION 3 CAMERA COMPUTER GET METHOD CALIBRATIONS LIST CALL ERROR
               "716676" : Bool;   // (IS_SEOC) UNIT 1 STATION 3 CAMERA COMPUTER GET METHOD ANALISIS LIST CALL ERROR
               "716677" : Bool;   // (IS_SEOC) UNIT 1 STATION 3 CAMERA COMPUTER RELEASE HANDLE LIST CALL ERROR
               "716678" : Bool;   // (IS_SEOC) UNIT 1 STATION 3 CAMERA COMPUTER RELEASE METHOD HANDLE LIST CALL ERROR
               "716679" : Bool;   // (IS_SEOC) UNIT 1 STATION 3 CAMERA COMPUTER DISCONNECT CALL ERROR
               "716680" : Bool;   // (IS_SEOC) UNIT 1 STATION 3 CAMERA COMPUTER DISCONNECT ALARM
               "716720" : Bool;   // (IS_SEOC) UNIT 1 STATION 3 COAXIAL CAMERA START LASER CALIBRATION METHOD CONNECTION ALARM
               "716721" : Bool;   // (IS_SEOC) UNIT 1 STATION 3 COAXIAL CAMERA START LASER CALIBRATION METHOD WORKING OR BLOCKED ALARM
               "716728" : Bool;   // (IS_SEOC) UNIT 1 STATION 3 COAXIAL CAMERA START NOZZLE CALIBRATION METHOD CONNECTION ALARM
               "716729" : Bool;   // (IS_SEOC) UNIT 1 STATION 3 COAXIAL CAMERA START NOZZLE CALIBRATION METHOD WORKING OR BLOCKED ALARM
               "716736" : Bool;   // (IS_SEOC) UNIT 1 STATION 3 COAXIAL CAMERA START JET CALIBRATION METHOD CONNECTION ALARM
               "716737" : Bool;   // (IS_SEOC) UNIT 1 STATION 3 COAXIAL CAMERA START JET CALIBRATION METHOD WORKING OR BLOCKED ALARM
               "716744" : Bool;   // (IS_SEOC) UNIT 1 STATION 3 COAXIAL CAMERA START CLADDING CALIBRATION METHOD CONNECTION ALARM
               "716745" : Bool;   // (IS_SEOC) UNIT 1 STATION 3 COAXIAL CAMERA START CLADDING CALIBRATION METHOD WORKING OR BLOCKED ALARM
               "716752" : Bool;   // (IS_SEOC) UNIT 1 STATION 3 COAXIAL CAMERA START NOZZLE ANALISIS METHOD CONNECTION ALARM
               "716753" : Bool;   // (IS_SEOC) UNIT 1 STATION 3 COAXIAL CAMERA START NOZZLE ANALISIS METHOD WORKING OR BLOCKED ALARM
               "716760" : Bool;   // (IS_SEOC) UNIT 1 STATION 3 COAXIAL CAMERA START JET ANALISIS METHOD CONNECTION ALARM
               "716761" : Bool;   // (IS_SEOC) UNIT 1 STATION 3 COAXIAL CAMERA START JET ANALISIS METHOD WORKING OR BLOCKED ALARM
               "716768" : Bool;   // (IS_SEOC) UNIT 1 STATION 3 COAXIAL CAMERA START CLADDING ANALISIS METHOD CONNECTION ALARM
               "716769" : Bool;   // (IS_SEOC) UNIT 1 STATION 3 COAXIAL CAMERA START CLADDING ANALISIS METHOD WORKING OR BLOCKED ALARM
               "716776" : Bool;   // (IS_SEOC) UNIT 1 STATION 3 COAXIAL CAMERA STOP METHODS CONNECTION ALARM
               "716777" : Bool;   // (IS_SEOC) UNIT 1 STATION 3 COAXIAL CAMERA STOP METHODS METHOD WORKING OR BLOCKED ALARM
               "716784" : Bool;   // (IS_SEOC) UNIT 1 STATION 3 COAXIAL CAMERA RESET PC METHOD CONNECTION ALARM
               "716785" : Bool;   // (IS_SEOC) UNIT 1 STATION 3 COAXIAL CAMERA RESET PC METHOD WORKING OR BLOCKED ALARM
               "716792" : Bool;   // (IS_SEOC) UNIT 1 STATION 3 COAXIAL CAMERA READ VARIABLES METHOD CONNECTION ALARM
               "716793" : Bool;   // (IS_SEOC) UNIT 1 STATION 3 COAXIAL CAMERA READ VARIABLES METHOD WORKING OR BLOCKED ALARM
            END_STRUCT;
         END_STRUCT;
         UNIT_02 : Struct   // UNIT 02 ALARMS
            "720000" : Bool;   // (IS_SEOC) UNIT 2 FIXTURE 1 PART TYPE DISCORDANCY ALARM
            "720001" : Bool;   // (IS_SEOC) UNIT 2 FIXTURE 2 PART TYPE DISCORDANCY ALARM
            "720002" : Bool;   // (IS_SEOC) UNIT 2 FIXTURE 3 PART TYPE DISCORDANCY ALARM
            "720003" : Bool;   // (IS_SEOC) UNIT 2 FIXTURE 4 PART TYPE DISCORDANCY ALARM
            "720008" : Bool;   // (RHP_SEOC) UNIT 2 FIXTURE 1 PART PRESENT DISCORDANCY ALARM
            "720009" : Bool;   // (RHP_SEOC) UNIT 2 FIXTURE 2 PART PRESENT DISCORDANCY ALARM
            "720010" : Bool;   // (RHP_SEOC) UNIT 2 FIXTURE 3 PART PRESENT DISCORDANCY ALARM
            "720011" : Bool;   // (RHP_SEOC) UNIT 2 FIXTURE 4 PART PRESENT DISCORDANCY ALARM
            "720024" : Bool;   // (IS_SEOC) UNIT 2 FIXTURE 1 PART ORIENTATION DISCORDANCY ALARM
            "720025" : Bool;   // (IS_SEOC) UNIT 2 FIXTURE 2 PART ORIENTATION DISCORDANCY ALARM
            "720026" : Bool;   // (IS_SEOC) UNIT 2 FIXTURE 3 PART ORIENTATION DISCORDANCY ALARM
            "720027" : Bool;   // (IS_SEOC) UNIT 2 FIXTURE 4 PART ORIENTATION DISCORDANCY ALARM
            "720032" : Bool;   // (RHP_SEOC) UNIT 2 FIXTURE 1 NOT CLAMPED DURING MACHINING ALARM
            "720033" : Bool;   // (RHP_SEOC) UNIT 2 FIXTURE 2 NOT CLAMPED DURING MACHINING ALARM
            "720034" : Bool;   // (RHP_SEOC) UNIT 2 FIXTURE 3 NOT CLAMPED DURING MACHINING ALARM
            "720035" : Bool;   // (RHP_SEOC) UNIT 2 FIXTURE 4 NOT CLAMPED DURING MACHINING ALARM
            STATION_2_MEASURING : Struct   // STATION 2 MEASURING ALARMS
               "720480" : Bool;   // (IS_SEOC) UNIT 2 STATION 2 MEASURING LAST CALIBRATION OUT OF RANGE IN FIXTURE 1 ALARM
               "720481" : Bool;   // (IS_SEOC) UNIT 2 STATION 2 MEASURING LAST CALIBRATION OUT OF RANGE IN FIXTURE 2 ALARM
               "720482" : Bool;   // (IS_SEOC) UNIT 2 STATION 2 MEASURING LAST CALIBRATION OUT OF RANGE IN FIXTURE 3 ALARM
               "720483" : Bool;   // (IS_SEOC) UNIT 2 STATION 2 MEASURING LAST CALIBRATION OUT OF RANGE IN FIXTURE 4 ALARM
               "720488" : Bool;   // (IS_SEOC) UNIT 2 STATION 2 MEASURING COMPUTER CONNECTION CALL ERROR
               "720489" : Bool;   // (IS_SEOC) UNIT 2 STATION 2 MEASURING COMPUTER GET INDEX LIST CALL ERROR
               "720490" : Bool;   // (IS_SEOC) UNIT 2 STATION 2 MEASURING COMPUTER GET HANDLE LIST CALL ERROR
               "720491" : Bool;   // (IS_SEOC) UNIT 2 STATION 2 MEASURING COMPUTER GET METHOD LIST CALL ERROR
               "720492" : Bool;   // (IS_SEOC) UNIT 2 STATION 2 MEASURING COMPUTER RELEASE HANDLE LIST CALL ERROR
               "720493" : Bool;   // (IS_SEOC) UNIT 2 STATION 2 MEASURING COMPUTER RELEASE METHOD HANDLE LIST CALL ERROR
               "720494" : Bool;   // (IS_SEOC) UNIT 2 STATION 2 MEASURING COMPUTER DISCONNECT CALL ERROR
               "720500" : Bool;   // (IS_SEOC) UNIT 2 STATION 2 MEASURING COMPUTER ERROR: PROFILER CONFIGURATION (ISSUES WITH THE PROFILOMETER CONFIGURATION)
               "720501" : Bool;   // (IS_SEOC) UNIT 2 STATION 2 MEASURING COMPUTER ERROR: ANALYZER CONFIGURATION (ERROR OCCURRED WHILE VERIFYING THE CONFIGURATION FILES)
               "720502" : Bool;   // (IS_SEOC) UNIT 2 STATION 2 MEASURING COMPUTER ERROR: DMC STRUCTURE (PROBLEMS READING THE DMC STRING)
               "720503" : Bool;   // (IS_SEOC) UNIT 2 STATION 2 MEASURING COMPUTER ERROR: ACQUISITION (UNABLE TO ACQUIRE PROFILES FROM THE PROFILOMETER)
               "720504" : Bool;   // (IS_SEOC) UNIT 2 STATION 2 MEASURING COMPUTER ERROR: PROFILE INITIALIZATION (FAILED TO INITIALIZE THE PROFILOMETER)
               "720505" : Bool;   // (IS_SEOC) UNIT 2 STATION 2 MEASURING COMPUTER ERROR: RUNOUT ANALYSIS (ISSUES EXECUTING THE RUNOUT ALGORITHM)
               "720506" : Bool;   // (IS_SEOC) UNIT 2 STATION 2 MEASURING COMPUTER ERROR: UMBRELLA ANALYSIS (ISSUES EXECUTING THE UMBRELLA ALGORITHM)
               "720508" : Bool;   // (IS_SEOC) UNIT 2 STATION 2 MEASURING COMPUTER ERROR: SURFACE DEFECTS ANALYSIS (ISSUES EXECUTING THE SURFACE DEFECTS ALGORITHM)
               "720509" : Bool;   // (IS_SEOC) UNIT 2 STATION 2 MEASURING COMPUTER ERROR: STORAGE ERROR (ERROR ATTEMPTING TO STORE DATA)
               "720510" : Bool;   // (IS_SEOC) UNIT 2 STATION 2 MEASURING COMPUTER ERROR: DATABASE CONNECTIN ALARM (CALIBRATION CHECK OR MEASURE SAVE NOT POSSIBLE)
               "720511" : Bool;   // (IS_SEOC) UNIT 2 STATION 2 MEASURING COMPUTER ERROR: CALIBRATION PROCEDURE (CALIBRATION FAILED)
               "720512" : Bool;   // (IS_SEOC) UNIT 2 STATION 2 MEASURING COMPUTER ERROR: CALIBRATION MISSING IN FIXTURE 1 (CALIBRATION MISSING OR FILE NOT FOUND)
               "720513" : Bool;   // (IS_SEOC) UNIT 2 STATION 2 MEASURING COMPUTER ERROR: CALIBRATION MISSING IN FIXTURE 2 (CALIBRATION MISSING OR FILE NOT FOUND)
               "720514" : Bool;   // (IS_SEOC) UNIT 2 STATION 2 MEASURING COMPUTER ERROR: CALIBRATION MISSING IN FIXTURE 3 (CALIBRATION MISSING OR FILE NOT FOUND)
               "720515" : Bool;   // (IS_SEOC) UNIT 2 STATION 2 MEASURING COMPUTER ERROR: CALIBRATION MISSING IN FIXTURE 4 (CALIBRATION MISSING OR FILE NOT FOUND)
               "720516" : Bool;   // (IS_SEOC) UNIT 2 STATION 2 MEASURING COMPUTER ERROR: PLC-PC MAJOR VERSIONS MISMATCH
               "720517" : Bool;   // (SEOC) UNIT 2 STATION 2 MEASURING COMPUTER ERROR: INITIALIZING PROFILOMETER
               "720530" : Bool;   // (IS_SEOC) UNIT 2 STATION 2 MEASURING COMPUTER MEASURING METHOD CALL EXECUTION ERROR
               "720531" : Bool;   // (IS_SEOC) UNIT 2 STATION 2 MEASURING COMPUTER MEASURING METHOD WORKING OR BLOCKED ERROR
               "720538" : Bool;   // (IS_SEOC) UNIT 2 STATION 2 MEASURING COMPUTER CALIBRATING METHOD CALL EXECUTION ERROR
               "720539" : Bool;   // (IS_SEOC) UNIT 2 STATION 2 MEASURING COMPUTER CALIBRATING METHOD WORKING OR BLOCKED ERROR
               "720546" : Bool;   // (IS_SEOC) UNIT 2 STATION 2 MEASURING COMPUTER RESET METHOD CALL EXECUTION ERROR
               "720547" : Bool;   // (IS_SEOC) UNIT 2 STATION 2 MEASURING COMPUTER RESET METHOD WORKING OR BLOCKED ERROR
               "720554" : Bool;   // (IS_SEOC) UNIT 2 STATION 2 MEASURING COMPUTER READ VARIABLES METHOD CALL EXECUTION ERROR
               "720555" : Bool;   // (IS_SEOC) UNIT 2 STATION 2 MEASURING COMPUTER READ VARIABLES METHOD WORKING OR BLOCKED ERROR
            END_STRUCT;
            STATION_3_MEASURING : Struct   // STATION 3 MEASURING ALARMS
               "720640" : Bool;   // (IS_SEOC) UNIT 2 STATION 3 MEASURING LAST CALIBRATION OUT OF RANGE IN FIXTURE 1 ALARM
               "720641" : Bool;   // (IS_SEOC) UNIT 2 STATION 3 MEASURING LAST CALIBRATION OUT OF RANGE IN FIXTURE 2 ALARM
               "720642" : Bool;   // (IS_SEOC) UNIT 2 STATION 3 MEASURING LAST CALIBRATION OUT OF RANGE IN FIXTURE 3 ALARM
               "720643" : Bool;   // (IS_SEOC) UNIT 2 STATION 3 MEASURING LAST CALIBRATION OUT OF RANGE IN FIXTURE 4 ALARM
               "720660" : Bool;   // (IS_SEOC) UNIT 2 STATION 3 MEASURING COMPUTER ERROR: PROFILER CONFIGURATION (ISSUES WITH THE PROFILOMETER CONFIGURATION)
               "720661" : Bool;   // (IS_SEOC) UNIT 2 STATION 3 MEASURING COMPUTER ERROR: ANALYZER CONFIGURATION (ERROR OCCURRED WHILE VERIFYING THE CONFIGURATION FILES)
               "720662" : Bool;   // (IS_SEOC) UNIT 2 STATION 3 MEASURING COMPUTER ERROR: DMC STRUCTURE (PROBLEMS READING THE DMC STRING)
               "720663" : Bool;   // (IS_SEOC) UNIT 2 STATION 3 MEASURING COMPUTER ERROR: ACQUISITION (UNABLE TO ACQUIRE PROFILES FROM THE PROFILOMETER)
               "720664" : Bool;   // (IS_SEOC) UNIT 2 STATION 3 MEASURING COMPUTER ERROR: PROFILE INITIALIZATION (FAILED TO INITIALIZE THE PROFILOMETER)
               "720665" : Bool;   // (IS_SEOC) UNIT 2 STATION 3 MEASURING COMPUTER ERROR: DISTANCE CALCULATION (ISSUES EXECUTING THE DISTANCE CALCULATION ALGORITHM)
               "720666" : Bool;   // (IS_SEOC) UNIT 2 STATION 3 MEASURING COMPUTER ERROR: LAYER GROWTH ANALYSIS (ISSUES EXECUTING THE LAYER GROWTH ALGORITHM)
               "720667" : Bool;   // (IS_SEOC) UNIT 2 STATION 3 MEASURING COMPUTER ERROR: STORAGE ERROR (ERROR ATTEMPTING TO STORE DATA)
               "720668" : Bool;   // (IS_SEOC) UNIT 2 STATION 3 MEASURING COMPUTER ERROR: DATABASE CONNECTION ALARM (CALIBRATION CHECK OR MEASURE SAVE NOT POSSIBLE)
               "720669" : Bool;   // (IS_SEOC) UNIT 2 STATION 3 MEASURING COMPUTER ERROR: CALIBRATION PROCEDURE (CALIBRATION FAILED)
               "720670" : Bool;   // (IS_SEOC) UNIT 2 STATION 3 MEASURING COMPUTER ERROR: CALIBRATION MISSING IN FIXTURE 1 (CALIBRATION MISSING OR FILE NOT FOUND)
               "720671" : Bool;   // (IS_SEOC) UNIT 2 STATION 3 MEASURING COMPUTER ERROR: CALIBRATION MISSING IN FIXTURE 2 (CALIBRATION MISSING OR FILE NOT FOUND)
               "720672" : Bool;   // (IS_SEOC) UNIT 2 STATION 3 MEASURING COMPUTER ERROR: CALIBRATION MISSING IN FIXTURE 3 (CALIBRATION MISSING OR FILE NOT FOUND)
               "720673" : Bool;   // (IS_SEOC) UNIT 2 STATION 3 MEASURING COMPUTER ERROR: CALIBRATION MISSING IN FIXTURE 4 (CALIBRATION MISSING OR FILE NOT FOUND)
               "720674" : Bool;   // (IS_SEOC) UNIT 2 STATION 3 MEASURING COMPUTER ERROR: PLC-PC MAJOR VERSIONS MISMATCH
               "720675" : Bool;   // (SEOC) UNIT 2 STATION 3 MEASURING COMPUTER ERROR: INITIALIZING PROFILOMETER
               "720680" : Bool;   // (IS_SEOC) UNIT 2 STATION 3 MEASURING COMPUTER NOZZLE SURFACE DISTANCE UPDATE ALARM
               "720688" : Bool;   // (IS_SEOC) UNIT 2 STATION 3 MEASURING COMPUTER CONNECTION ALARM
               "720689" : Bool;   // (IS_SEOC) UNIT 2 STATION 3 MEASURING COMPUTER GET INDEX LIST ALARM
               "720690" : Bool;   // (IS_SEOC) UNIT 2 STATION 3 MEASURING COMPUTER START NOOZLE MEASUREMENT METHOD CALL EXECUTION ERROR
               "720691" : Bool;   // (IS_SEOC) UNIT 2 STATION 3 MEASURING COMPUTER START NOOZLE MEASUREMENT METHOD WORKING OR BLOCKED ERROR
               "720692" : Bool;   // (IS_SEOC) UNIT 2 STATION 3 MEASURING COMPUTER RELEASE HANDLE LIST ALARM
               "720693" : Bool;   // (IS_SEOC) UNIT 2 STATION 3 MEASURING COMPUTER RELEASE METHOD LIST ALARM
               "720694" : Bool;   // (IS_SEOC) UNIT 2 STATION 3 MEASURING COMPUTER DISCONNECT ALARM
               "720706" : Bool;   // (IS_SEOC) UNIT 2 STATION 3 MEASURING COMPUTER START LAYER THICKNESS MEASUREMENT METHOD CALL EXECUTION ERROR
               "720707" : Bool;   // (IS_SEOC) UNIT 2 STATION 3 MEASURING COMPUTER START LAYER THICKNESS MEASUREMENT METHOD WORKING OR BLOCKED ERROR
               "720714" : Bool;   // (IS_SEOC) UNIT 2 STATION 3 MEASURING COMPUTER STOP LAYER THICKNESS MEASUREMENT METHOD CALL EXECUTION ERROR
               "720715" : Bool;   // (IS_SEOC) UNIT 2 STATION 3 MEASURING COMPUTER STOP LAYER THICKNESS MEASUREMENT METHOD WORKING OR BLOCKED ERROR
               "720722" : Bool;   // (IS_SEOC) UNIT 2 STATION 3 MEASURING COMPUTER CALIBRATING METHOD CALL EXECUTION ERROR
               "720723" : Bool;   // (IS_SEOC) UNIT 2 STATION 3 MEASURING COMPUTER CALIBRATING METHOD WORKING OR BLOCKED ERROR
               "720730" : Bool;   // (IS_SEOC) UNIT 2 STATION 3 MEASURING COMPUTER RESET METHOD CALL EXECUTION ERROR
               "720731" : Bool;   // (IS_SEOC) UNIT 2 STATION 3 MEASURING COMPUTER RESET METHOD WORKING OR BLOCKED ERROR
               "720738" : Bool;   // (IS_SEOC) UNIT 2 STATION 3 MEASURING COMPUTER READ VARIABLES METHOD CALL EXECUTION ERROR
               "720739" : Bool;   // (IS_SEOC) UNIT 2 STATION 3 MEASURING COMPUTER READ VARIABLES METHOD WORKING OR BLOCKED ERROR
            END_STRUCT;
            STATION_3_COAXIAL : Struct   // STATION 3 COAXIAL ALARMS
               "720800" : Bool;   // (IS_SEOC) UNIT 2 STATION 3 CAMERA COMPUTER ERROR: FAILED TO CONNECT TO CAMERA (UNABLE TO GET IMAGES FROM CAMERA)
               "720801" : Bool;   // (IS_SEOC) UNIT 2 STATION 3 CAMERA COMPUTER ERROR: FAILED TO SET CAMERA PARAMETERS (UNABLE TO SET CAMERA PARAMETERS (EXPOSURE-TIME & GAIN) FROM CURRENT IMAGES)
               "720802" : Bool;   // (IS_SEOC) UNIT 2 STATION 3 CAMERA COMPUTER ERROR: NEW LASER CALIBRATION REQUIERED (CURRENT CALIBRATION PARAMETERS DO NOT MEEST RECENT ANALYSIS REQUISITES)
               "720804" : Bool;   // (IS_SEOC) UNIT 2 STATION 3 CAMERA COMPUTER ERROR: NEW JET CALIBRATION REQUIERED (CURRENT CALIBRATION PARAMETERS DO NOT MEEST RECENT ANALYSIS REQUISITES)
               "720805" : Bool;   // (IS_SEOC) UNIT 2 STATION 3 CAMERA COMPUTER ERROR: NEW CLADDING CALIBRATION REQUIERED (CURRENT CALIBRATION PARAMETERS DO NOT MEEST RECENT ANALYSIS REQUISITES)
               "720806" : Bool;   // (IS_SEOC) UNIT 2 STATION 3 CAMERA COMPUTER ERROR: HIGH NUMBER OF DEAD PIXELS (THE NUMBER OF DEAD-PIXELS EXCEEDS A CONFIGURED NUMBER)
               "720807" : Bool;   // (IS_SEOC) UNIT 2 STATION 3 CAMERA COMPUTER ERROR: NO LIGHT DETECTED (NO LIGHT OR BLANK IMAGE DETECTED)
               "720808" : Bool;   // (IS_SEOC) UNIT 2 STATION 3 CAMERA COMPUTER ERROR: NO LASER DETECTED (NO LASER SPOT DETECTED)
               "720809" : Bool;   // (IS_SEOC) UNIT 2 STATION 3 CAMERA COMPUTER ERROR: NO NOZZLE DETECTED (UNABLE TO DETECT ANY CAPSULE-SHAPED NOZZLE IN THE IMAGE)
               "720810" : Bool;   // (IS_SEOC) UNIT 2 STATION 3 CAMERA COMPUTER ERROR: NO POWDER FLOW DETECTED (NO POWDER FLOW HAS BEEN DETECTED IN THE IMAGE)
               "720811" : Bool;   // (IS_SEOC) UNIT 2 STATION 3 CAMERA COMPUTER ERROR: NO LASER PATERN DETECTED (NO LASER PATERN HAS BEEN DETECTED IN THE IMAGE)
               "720812" : Bool;   // (IS_SEOC) UNIT 2 STATION 3 CAMERA COMPUTER ERROR: NOT ANALYZED
               "720813" : Bool;   // (IS_SEOC) UNIT 2 STATION 3 CAMERA COMPUTER ERROR: FAILED TO OBTAIN SCALE FACTOR
               "720814" : Bool;   // (IS_SEOC) UNIT 2 STATION 3 CAMERA COMPUTER ERROR: UNALIGNED POWDER FLOW VORTEX
               "720815" : Bool;   // (IS_SEOC) UNIT 2 STATION 3 CAMERA COMPUTER ERROR: JET MALFUNCTION
               "720816" : Bool;   // (IS_SEOC) UNIT 2 STATION 3 CAMERA COMPUTER ERROR: UNCALIBRATED
               "720817" : Bool;   // (IS_SEOC) UNIT 2 STATION 3 CAMERA COMPUTER ERROR: PLC-PC MAJOR VERSIONS MISMATCH
               "720818" : Bool;   // (IS_SEOC) UNIT 2 STATION 3 CAMERA COMPUTER ERROR: NO MELT POOL DETECTED
               "720819" : Bool;   // (IS_SEOC) UNIT 2 STATION 3 CAMERA COMPUTER ERROR: NO DATA VASE CONNECTION
               "720820" : Bool;   // (IS_SEOC) UNIT 2 STATION 3 CAMERA COMPUTER ERROR: NO HALO DETECTED
               "720821" : Bool;   // (IS_SEOC) UNIT 2 STATION 3 CAMERA COMPUTER ERROR: STORAGE ERROR
               "720822" : Bool;   // (SEOC) UNIT 2 STATION 3 CAMERA COMPUTER ERROR: INITIALIZING CAMERA
               "720823" : Bool;   // (IS_SEOC) UNIT 2 STATION 3 CAMERA COMPUTER ERROR: NOZZLE CONTAMINATION DETECTED
               "720824" : Bool;   // (IS_SEOC) UNIT 2 STATION 3 CAMERA COMPUTER ERROR: INVALID CONFIGURATION
               "720832" : Bool;   // (IS_SEOC) UNIT 2 STATION 3 CAMERA COMPUTER CONNECTION CALL ERROR
               "720833" : Bool;   // (IS_SEOC) UNIT 2 STATION 3 CAMERA COMPUTER GET INDEX LIST CALL ERROR
               "720834" : Bool;   // (IS_SEOC) UNIT 2 STATION 3 CAMERA COMPUTER GET HANDLE LIST CALL ERROR
               "720835" : Bool;   // (IS_SEOC) UNIT 2 STATION 3 CAMERA COMPUTER GET METHOD CALIBRATIONS LIST CALL ERROR
               "720836" : Bool;   // (IS_SEOC) UNIT 2 STATION 3 CAMERA COMPUTER GET METHOD ANALISIS LIST CALL ERROR
               "720837" : Bool;   // (IS_SEOC) UNIT 2 STATION 3 CAMERA COMPUTER RELEASE HANDLE LIST CALL ERROR
               "720838" : Bool;   // (IS_SEOC) UNIT 2 STATION 3 CAMERA COMPUTER RELEASE METHOD HANDLE LIST CALL ERROR
               "720839" : Bool;   // (IS_SEOC) UNIT 2 STATION 3 CAMERA COMPUTER DISCONNECT CALL ERROR
               "720880" : Bool;   // (IS_SEOC) UNIT 2 STATION 3 COAXIAL CAMERA START LASER CALIBRATION METHOD CONNECTION ALARM
               "720881" : Bool;   // (IS_SEOC) UNIT 2 STATION 3 COAXIAL CAMERA START LASER CALIBRATION METHOD WORKING OR BLOCKED ALARM
               "720888" : Bool;   // (IS_SEOC) UNIT 2 STATION 3 COAXIAL CAMERA START NOZZLE CALIBRATION METHOD CONNECTION ALARM
               "720889" : Bool;   // (IS_SEOC) UNIT 2 STATION 3 COAXIAL CAMERA START NOZZLE CALIBRATION METHOD WORKING OR BLOCKED ALARM
               "720896" : Bool;   // (IS_SEOC) UNIT 2 STATION 3 COAXIAL CAMERA START JET CALIBRATION METHOD CONNECTION ALARM
               "720897" : Bool;   // (IS_SEOC) UNIT 2 STATION 3 COAXIAL CAMERA START JET CALIBRATION METHOD WORKING OR BLOCKED ALARM
               "720904" : Bool;   // (IS_SEOC) UNIT 2 STATION 3 COAXIAL CAMERA START CLADDING CALIBRATION METHOD CONNECTION ALARM
               "720905" : Bool;   // (IS_SEOC) UNIT 2 STATION 3 COAXIAL CAMERA START CLADDING CALIBRATION METHOD WORKING OR BLOCKED ALARM
               "720912" : Bool;   // (IS_SEOC) UNIT 2 STATION 3 COAXIAL CAMERA START NOZZLE ANALISIS METHOD CONNECTION ALARM
               "720913" : Bool;   // (IS_SEOC) UNIT 2 STATION 3 COAXIAL CAMERA START NOZZLE ANALISIS METHOD WORKING OR BLOCKED ALARM
               "720920" : Bool;   // (IS_SEOC) UNIT 2 STATION 3 COAXIAL CAMERA START JET ANALISIS METHOD CONNECTION ALARM
               "720921" : Bool;   // (IS_SEOC) UNIT 2 STATION 3 COAXIAL CAMERA START JET ANALISIS METHOD WORKING OR BLOCKED ALARM
               "720928" : Bool;   // (IS_SEOC) UNIT 2 STATION 3 COAXIAL CAMERA START CLADDING ANALISIS METHOD CONNECTION ALARM
               "720929" : Bool;   // (IS_SEOC) UNIT 2 STATION 3 COAXIAL CAMERA START CLADDING ANALISIS METHOD WORKING OR BLOCKED ALARM
               "720936" : Bool;   // (IS_SEOC) UNIT 2 STATION 3 COAXIAL CAMERA STOP METHODS CONNECTION ALARM
               "720937" : Bool;   // (IS_SEOC) UNIT 2 STATION 3 COAXIAL CAMERA STOP METHODS METHOD WORKING OR BLOCKED ALARM
               "720944" : Bool;   // (IS_SEOC) UNIT 2 STATION 3 COAXIAL CAMERA REST PC METHOD CONNECTION ALARM
               "720945" : Bool;   // (IS_SEOC) UNIT 2 STATION 3 COAXIAL CAMERA REST PC METHOD WORKING OR BLOCKED ALARM
               "720952" : Bool;   // (IS_SEOC) UNIT 2 STATION 3 COAXIAL CAMERA READ VARIABLES METHOD CONNECTION ALARM
               "720953" : Bool;   // (IS_SEOC) UNIT 2 STATION 3 COAXIAL CAMERA READ VARIABLES METHOD WORKING BLOCKED ALARM
            END_STRUCT;
         END_STRUCT;
         UNIT_03 : Struct   // UNIT 03 ALARMS
            FACE_R_MEASURING : Struct   // FACE R MEASURING ALARMS
               "724240" : Bool;   // (IS_SEOC) MEASURING STATION COMPUTER FACE R ERROR: PROFILER CONFIGURATION (ISSUES WITH THE PROFILOMETER CONFIGURATION)
               "724241" : Bool;   // (IS_SEOC) MEASURING STATION COMPUTER FACE R ERROR: ANALYZER CONFIGURATION (ERROR OCCURRED WHILE VERIFYING THE CONFIGURATION FILES)
               "724242" : Bool;   // (IS_SEOC) MEASURING STATION COMPUTER FACE R ERROR: DMC STRUCTURE (PROBLEMS READING THE DMC STRING)
               "724243" : Bool;   // (IS_SEOC) MEASURING STATION COMPUTER FACE R ERROR: ACQUISITION (UNABLE TO ACQUIRE PROFILES FROM THE PROFILOMETER)
               "724244" : Bool;   // (IS_SEOC) MEASURING STATION COMPUTER FACE R ERROR: PROFILE INITIALIZATION (FAILED TO INITIALIZE THE PROFILOMETER)
               "724245" : Bool;   // (IS_SEOC) MEASURING STATION COMPUTER FACE R ERROR: RUNOUT ANALYSIS (ISSUES EXECUTING THE RUNOUT ALGORITHM)
               "724246" : Bool;   // (IS_SEOC) MEASURING STATION COMPUTER FACE R ERROR: UMBRELLA ANALYSIS (ISSUES EXECUTING THE UMBRELLA ALGORITHM)
               "724247" : Bool;   // (IS_SEOC) MEASURING STATION COMPUTER FACE R ERROR: LAYER GROWTH ANALYSIS (ISSUES EXECUTING THE LAYER GROWTH ALGORITHM)
               "724248" : Bool;   // (IS_SEOC) MEASURING STATION COMPUTER FACE R ERROR: SURFACE DEFECTS ANALYSIS (ISSUES EXECUTING THE SURFACE DEFECTS ALGORITHM)
               "724249" : Bool;   // (IS_SEOC) MEASURING STATION COMPUTER FACE R ERROR: STORAGE ERROR (ERROR ATTEMPTING TO STORE DATA)
               "724250" : Bool;   // (IS_SEOC) MEASURING STATION COMPUTER FACE R ERROR: MISSING CALIBRATION (CALIBRATION MISSING OR FILE NOT FOUND)
               "724251" : Bool;   // (IS_SEOC) MEASURING STATION COMPUTER FACE R ERROR: CALIBRATION PROCEDURE (CALIBRATION FAILED)
               "724252" : Bool;   // (IS_SEOC) MEASURING STATION COMPUTER FACE R ERROR: DISTANCE CALCULATION (ISSUES EXECUTING THE DISTANCE CALCULATION)
               "724253" : Bool;   // (IS_SEOC) MEASURING STATION COMPUTER FACE R ERROR: DATABASE CONNECTION ALARM (CALIBRATION CHECK OR MEASURE SAVE NO POSSIBLE)
               "724254" : Bool;   // (IS_SEOC) MEASURING STATION COMPUTER ERROR: PLC-PC MAJOR VERSIONS MISMATCH
               "724255" : Bool;   // (SEOC) MEASURING STATION COMPUTER ERROR: INITIALIZING PROFILOMETER
               "724260" : Bool;   // (IS_SEOC) MEASURING STATION COMPUTER FACE R MEASURING METHOD CALL EXECUTION ERROR
               "724261" : Bool;   // (IS_SEOC) MEASURING STATION COMPUTER FACE R MEASURING METHOD WORKING OR BLOCKED ERROR
               "724268" : Bool;   // (IS_SEOC) MEASURING STATION COMPUTER FACE R CALIBRATING METHOD CALL EXECUTION ERROR
               "724269" : Bool;   // (IS_SEOC) MEASURING STATION COMPUTER FACE R CALIBRATING METHOD WORKING OR BLOCKED ERROR
               "724276" : Bool;   // (IS_SEOC) MEASURING STATION COMPUTER FACE R RESET METHOD CALL EXECUTION ERROR
               "724277" : Bool;   // (IS_SEOC) MEASURING STATION COMPUTER FACE R RESET METHOD WORKING OR BLOCKED ERROR
               "724284" : Bool;   // (IS_SEOC) MEASURING STATION COMPUTER FACE R VARIABLE READING CALL CONEXION ERROR
               "724285" : Bool;   // (IS_SEOC) MEASURING STATION COMPUTER FACE R VARIABLE READING WORKING OR BLOCKED ERROR
               "724296" : Bool;   // (IS_SEOC) MEASURING STATION COMPUTER FACE R CONNECTION CALL ERROR
               "724297" : Bool;   // (IS_SEOC) MEASURING STATION COMPUTER FACE R GET INDEX LIST CALL ERROR
               "724298" : Bool;   // (IS_SEOC) MEASURING STATION COMPUTER FACE R GET HANDLE LIST CALL ERROR
               "724299" : Bool;   // (IS_SEOC) MEASURING STATION COMPUTER FACE R GET METHOD LIST CALL ERROR
               "724300" : Bool;   // (IS_SEOC) MEASURING STATION COMPUTER FACE R RELEASE HANDLE LIST CALL ERROR
               "724301" : Bool;   // (IS_SEOC) MEASURING STATION COMPUTER FACE R RELEASE METHOD HANDLE LIST CALL ERROR
               "724302" : Bool;   // (IS_SEOC) MEASURING STATION COMPUTER FACE R DISCONNECT CALL ERROR
            END_STRUCT;
            FACE_N_MEASURING : Struct   // FACE N MEASURING ALARMS
               "724400" : Bool;   // (IS_SEOC) MEASURING STATION COMPUTER FACE N ERROR: PROFILER CONFIGURATION (ISSUES WITH THE PROFILOMETER CONFIGURATION)
               "724401" : Bool;   // (IS_SEOC) MEASURING STATION COMPUTER FACE N ERROR: ANALYZER CONFIGURATION (ERROR OCCURRED WHILE VERIFYING THE CONFIGURATION FILES)
               "724402" : Bool;   // (IS_SEOC) MEASURING STATION COMPUTER FACE N ERROR: DMC STRUCTURE (PROBLEMS READING THE DMC STRING)
               "724403" : Bool;   // (IS_SEOC) MEASURING STATION COMPUTER FACE N ERROR: ACQUISITION (UNABLE TO ACQUIRE PROFILES FROM THE PROFILOMETER)
               "724404" : Bool;   // (IS_SEOC) MEASURING STATION COMPUTER FACE N ERROR: PROFILE INITIALIZATION (FAILED TO INITIALIZE THE PROFILOMETER)
               "724405" : Bool;   // (IS_SEOC) MEASURING STATION COMPUTER FACE N ERROR: RUNOUT ANALYSIS (ISSUES EXECUTING THE RUNOUT ALGORITHM)
               "724406" : Bool;   // (IS_SEOC) MEASURING STATION COMPUTER FACE N ERROR: UMBRELLA ANALYSIS (ISSUES EXECUTING THE UMBRELLA ALGORITHM)
               "724407" : Bool;   // (IS_SEOC) MEASURING STATION COMPUTER FACE N ERROR: LAYER GROWTH ANALYSIS (ISSUES EXECUTING THE LAYER GROWTH ALGORITHM)
               "724408" : Bool;   // (IS_SEOC) MEASURING STATION COMPUTER FACE N ERROR: SURFACE DEFECTS ANALYSIS (ISSUES EXECUTING THE SURFACE DEFECTS ALGORITHM)
               "724409" : Bool;   // (IS_SEOC) MEASURING STATION COMPUTER FACE N ERROR: STORAGE ERROR (ERROR ATTEMPTING TO STORE DATA)
               "724410" : Bool;   // (IS_SEOC) MEASURING STATION COMPUTER FACE N ERROR: MISSING CALIBRATION (CALIBRATION MISSING OR FILE NOT FOUND)
               "724411" : Bool;   // (IS_SEOC) MEASURING STATION COMPUTER FACE N ERROR: CALIBRATION PROCEDURE (CALIBRATION FAILED)
               "724412" : Bool;   // (IS_SEOC) MEASURING STATION COMPUTER FACE N ERROR: DISTANCE CALCULATION (ISSUES EXECUTING THE DISTANCE CALCULATION)
               "724413" : Bool;   // (IS_SEOC) MEASURING STATION COMPUTER FACE N ERROR: DATABASE CONNECTION ALARM (CALIBRATION CHECK OR MEASURE SAVE NO POSSIBLE)
               "724414" : Bool;   // (SEOC) MEASURING STATION COMPUTER ERROR: INITIALIZING PROFILOMETER
               "724420" : Bool;   // (IS_SEOC) MEASURING STATION COMPUTER FACE N MEASURING METHOD CALL EXECUTION ERROR
               "724421" : Bool;   // (IS_SEOC) MEASURING STATION COMPUTER FACE N MEASURING METHOD WORKING OR BLOCKED ERROR
               "724428" : Bool;   // (IS_SEOC) MEASURING STATION COMPUTER FACE N CALIBRATING METHOD CALL EXECUTION ERROR
               "724429" : Bool;   // (IS_SEOC) MEASURING STATION COMPUTER FACE N CALIBRATING METHOD WORKING OR BLOCKED ERROR
               "724436" : Bool;   // (IS_SEOC) MEASURING STATION COMPUTER FACE N RESET METHOD CALL EXECUTION ERROR
               "724437" : Bool;   // (IS_SEOC) MEASURING STATION COMPUTER FACE N RESET METHOD WORKING OR BLOCKED ERROR
               "724444" : Bool;   // (IS_SEOC) MEASURING STATION COMPUTER FACE N VARIABLE READING CALL CONEXION ERROR
               "724445" : Bool;   // (IS_SEOC) MEASURING STATION COMPUTER FACE N VARIABLE READING WORKING OR BLOCKED ERROR
               "724456" : Bool;   // (IS_SEOC) MEASURING STATION COMPUTER FACE N CONNECTION CALL ERROR
               "724457" : Bool;   // (IS_SEOC) MEASURING STATION COMPUTER FACE N GET INDEX LIST CALL ERROR
               "724458" : Bool;   // (IS_SEOC) MEASURING STATION COMPUTER FACE N GET HANDLE LIST CALL ERROR
               "724459" : Bool;   // (IS_SEOC) MEASURING STATION COMPUTER FACE N GET METHOD LIST CALL ERROR
               "724460" : Bool;   // (IS_SEOC) MEASURING STATION COMPUTER FACE N RELEASE HANDLE LIST CALL ERROR
               "724461" : Bool;   // (IS_SEOC) MEASURING STATION COMPUTER FACE N RELEASE METHOD HANDLE LIST CALL ERROR
               "724462" : Bool;   // (IS_SEOC) MEASURING STATION COMPUTER FACE N DISCONNECT CALL ERROR
            END_STRUCT;
         END_STRUCT;
         CYLINDERS : Struct   // CYLINDERS ALARMS
            "732001" : Bool;   // (IS_SEOC) UNIT 1 UP SEALING STRUCTURE CLOSED 1 INPUT ALARM
            "732002" : Bool;   // (IS_SEOC) UNIT 1 UP SEALING STRUCTURE CLOSED 2 INPUT ALARM
            "732003" : Bool;   // (IS_SEOC) UNIT 1 UP SEALING STRUCTURE CLOSED 3 INPUT ALARM
            "732004" : Bool;   // (IS_SEOC) UNIT 1 UP SEALING STRUCTURE CLOSED 4 INPUT ALARM
            "732011" : Bool;   // (IS_SEOC) UNIT 1 UP SEALING STRUCTURE OPENED 1 INPUT ALARM
            "732012" : Bool;   // (IS_SEOC) UNIT 1 UP SEALING STRUCTURE OPENED 2 INPUT ALARM
            "732013" : Bool;   // (IS_SEOC) UNIT 1 UP SEALING STRUCTURE OPENED 3 INPUT ALARM
            "732014" : Bool;   // (IS_SEOC) UNIT 1 UP SEALING STRUCTURE OPENED 4 INPUT ALARM
            "732021" : Bool;   // (IS_SEOC) UNIT 1 DOWN SEALING STRUCTURE CLOSED 1 INPUT ALARM
            "732022" : Bool;   // (IS_SEOC) UNIT 1 DOWN SEALING STRUCTURE CLOSED 2 INPUT ALARM
            "732023" : Bool;   // (IS_SEOC) UNIT 1 DOWN SEALING STRUCTURE CLOSED 3 INPUT ALARM
            "732024" : Bool;   // (IS_SEOC) UNIT 1 DOWN SEALING STRUCTURE CLOSED 4 INPUT ALARM
            "732031" : Bool;   // (IS_SEOC) UNIT 1 DOWN SEALING STRUCTURE OPENED 1 INPUT ALARM
            "732032" : Bool;   // (IS_SEOC) UNIT 1 DOWN SEALING STRUCTURE OPENED 2 INPUT ALARM
            "732033" : Bool;   // (IS_SEOC) UNIT 1 DOWN SEALING STRUCTURE OPENED 3 INPUT ALARM
            "732034" : Bool;   // (IS_SEOC) UNIT 1 DOWN SEALING STRUCTURE OPENED 4 INPUT ALARM
            "732361" : Bool;   // (IS_SEOC) UNIT 1 Z13 SAFETY BRAKE BLOCKED ALARM
            "732362" : Bool;   // (IS_SEOC) UNIT 1 Z13 SAFETY BRAKE UNBLOCKED ALARM
            "732363" : Bool;   // (IS_SEOC) UNIT 1 Z13 SAFETY BRAKE MAINTENANCE SENSORS ALARM
            "732380" : Bool;   // (IS_SEOC) UNIT 1 ANGULAR LOCATOR CYLINDER ADVANCED INPUT 1 ALARM
            "732381" : Bool;   // (IS_SEOC) UNIT 1 ANGULAR LOCATOR CYLINDER ADVANCED INPUT 2 ALARM
            "732382" : Bool;   // (IS_SEOC) UNIT 1 ANGULAR LOCATOR CYLINDER ADVANCED INPUT 3 ALARM
            "732383" : Bool;   // (IS_SEOC) UNIT 1 ANGULAR LOCATOR CYLINDER ADVANCED INPUT 4 ALARM
            "732390" : Bool;   // (IS_SEOC) UNIT 1 ANGULAR LOCATOR CYLINDER RETURNED INPUT 1 ALARM
            "732391" : Bool;   // (IS_SEOC) UNIT 1 ANGULAR LOCATOR CYLINDER RETURNED INPUT 2 ALARM
            "732392" : Bool;   // (IS_SEOC) UNIT 1 ANGULAR LOCATOR CYLINDER RETURNED INPUT 3 ALARM
            "732393" : Bool;   // (IS_SEOC) UNIT 1 ANGULAR LOCATOR CYLINDER RETURNED INPUT 4 ALARM
            "732410" : Bool;   // (IS_SEOC) UNIT 1 AXIAL LOCATOR CYLINDER ADVANCED INPUT 1 ALARM
            "732411" : Bool;   // (IS_SEOC) UNIT 1 AXIAL LOCATOR CYLINDER ADVANCED INPUT 2 ALARM
            "732412" : Bool;   // (IS_SEOC) UNIT 1 AXIAL LOCATOR CYLINDER ADVANCED INPUT 3 ALARM
            "732413" : Bool;   // (IS_SEOC) UNIT 1 AXIAL LOCATOR CYLINDER ADVANCED INPUT 4 ALARM
            "732420" : Bool;   // (IS_SEOC) UNIT 1 AXIAL LOCATOR CYLINDER RETURNED INPUT 1 ALARM
            "732421" : Bool;   // (IS_SEOC) UNIT 1 AXIAL LOCATOR CYLINDER RETURNED INPUT 2 ALARM
            "732422" : Bool;   // (IS_SEOC) UNIT 1 AXIAL LOCATOR CYLINDER RETURNED INPUT 3 ALARM
            "732423" : Bool;   // (IS_SEOC) UNIT 1 AXIAL LOCATOR CYLINDER RETURNED INPUT 4 ALARM
            "732721" : Bool;   // (IS_SEOC) UNIT 2 UP SEALING STRUCTURE CLOSED 1 INPUT ALARM
            "732722" : Bool;   // (IS_SEOC) UNIT 2 UP SEALING STRUCTURE CLOSED 2 INPUT ALARM
            "732723" : Bool;   // (IS_SEOC) UNIT 2 UP SEALING STRUCTURE CLOSED 3 INPUT ALARM
            "732724" : Bool;   // (IS_SEOC) UNIT 2 UP SEALING STRUCTURE CLOSED 4 INPUT ALARM
            "732731" : Bool;   // (IS_SEOC) UNIT 2 UP SEALING STRUCTURE OPENED 1 INPUT ALARM
            "732732" : Bool;   // (IS_SEOC) UNIT 2 UP SEALING STRUCTURE OPENED 2 INPUT ALARM
            "732733" : Bool;   // (IS_SEOC) UNIT 2 UP SEALING STRUCTURE OPENED 3 INPUT ALARM
            "732734" : Bool;   // (IS_SEOC) UNIT 2 UP SEALING STRUCTURE OPENED 4 INPUT ALARM
            "732741" : Bool;   // (IS_SEOC) UNIT 2 DOWN SEALING STRUCTURE CLOSED 1 INPUT ALARM
            "732742" : Bool;   // (IS_SEOC) UNIT 2 DOWN SEALING STRUCTURE CLOSED 2 INPUT ALARM
            "732743" : Bool;   // (IS_SEOC) UNIT 2 DOWN SEALING STRUCTURE CLOSED 3 INPUT ALARM
            "732744" : Bool;   // (IS_SEOC) UNIT 2 DOWN SEALING STRUCTURE CLOSED 4 INPUT ALARM
            "732751" : Bool;   // (IS_SEOC) UNIT 2 DOWN SEALING STRUCTURE OPENED 1 INPUT ALARM
            "732752" : Bool;   // (IS_SEOC) UNIT 2 DOWN SEALING STRUCTURE OPENED 2 INPUT ALARM
            "732753" : Bool;   // (IS_SEOC) UNIT 2 DOWN SEALING STRUCTURE OPENED 3 INPUT ALARM
            "732754" : Bool;   // (IS_SEOC) UNIT 2 DOWN SEALING STRUCTURE OPENED 4 INPUT ALARM
            "733081" : Bool;   // (IS_SEOC) UNIT 2 Z23 SAFETY BRAKE BLOCKED ALARM
            "733082" : Bool;   // (IS_SEOC) UNIT 2 Z23 SAFETY BRAKE UNBLOCKED ALARM
            "733083" : Bool;   // (IS_SEOC) UNIT 2 Z23 SAFETY BRAKE MAINTENANCE SENSORS ALARM
            "733100" : Bool;   // (IS_SEOC) UNIT 2 ANGULAR LOCATOR CYLINDER ADVANCED INPUT 1 ALARM
            "733101" : Bool;   // (IS_SEOC) UNIT 2 ANGULAR LOCATOR CYLINDER ADVANCED INPUT 2 ALARM
            "733102" : Bool;   // (IS_SEOC) UNIT 2 ANGULAR LOCATOR CYLINDER ADVANCED INPUT 3 ALARM
            "733103" : Bool;   // (IS_SEOC) UNIT 2 ANGULAR LOCATOR CYLINDER ADVANCED INPUT 4 ALARM
            "733110" : Bool;   // (IS_SEOC) UNIT 2 ANGULAR LOCATOR CYLINDER RETURNED INPUT 1 ALARM
            "733111" : Bool;   // (IS_SEOC) UNIT 2 ANGULAR LOCATOR CYLINDER RETURNED INPUT 2 ALARM
            "733112" : Bool;   // (IS_SEOC) UNIT 2 ANGULAR LOCATOR CYLINDER RETURNED INPUT 3 ALARM
            "733113" : Bool;   // (IS_SEOC) UNIT 2 ANGULAR LOCATOR CYLINDER RETURNED INPUT 4 ALARM
            "733130" : Bool;   // (IS_SEOC) UNIT 2 AXIAL LOCATOR CYLINDER ADVANCED INPUT 1 ALARM
            "733131" : Bool;   // (IS_SEOC) UNIT 2 AXIAL LOCATOR CYLINDER ADVANCED INPUT 2 ALARM
            "733132" : Bool;   // (IS_SEOC) UNIT 2 AXIAL LOCATOR CYLINDER ADVANCED INPUT 3 ALARM
            "733133" : Bool;   // (IS_SEOC) UNIT 2 AXIAL LOCATOR CYLINDER ADVANCED INPUT 4 ALARM
            "733140" : Bool;   // (IS_SEOC) UNIT 2 AXIAL LOCATOR CYLINDER RETURNED INPUT 1 ALARM
            "733141" : Bool;   // (IS_SEOC) UNIT 2 AXIAL LOCATOR CYLINDER RETURNED INPUT 2 ALARM
            "733142" : Bool;   // (IS_SEOC) UNIT 2 AXIAL LOCATOR CYLINDER RETURNED INPUT 3 ALARM
            "733143" : Bool;   // (IS_SEOC) UNIT 2 AXIAL LOCATOR CYLINDER RETURNED INPUT 4 ALARM
         END_STRUCT;
         LASER_SYSTEM : Struct   // LASER SYSTEM ALARMS
            "736000" : Bool;   // (RHP_SEOC) LASER UNIT 1 READY CIRCUIT BREAKER ALARM
            "736001" : Bool;   // (RHP_SEOC) LASER UNIT 1 READY LASER ERROR
            "736002" : Bool;   // (RHP_SEOC) LASER UNIT 1 READY WARNING LASER
            "736003" : Bool;   // (RHP_SEOC) LASER UNIT 1 READY LASER NOT READY
            "736004" : Bool;   // (RHP_SEOC) LASER UNIT 1 READY LASER NOT SWITCHED ON
            "736005" : Bool;   // (RHP_SEOC) LASER UNIT 1 READY ANALOG CONTROL ERROR
            "736006" : Bool;   // (RHP_SEOC) LASER UNIT 1 READY LASER NOT ASSIGNED
            "736007" : Bool;   // (RHP_SEOC) LASER UNIT 1 READY OVERTEMPERATURE ALARM
            "736008" : Bool;   // (RHP_SEOC) LASER UNIT 1 READY LASER EMERGENCY STOP ACTIVE
            "736009" : Bool;   // (RHP_SEOC) LASER UNIT 1 READY LASER SC STATUS ACTIVE
            "736010" : Bool;   // (RHP_SEOC) LASER UNIT 1 READY ACTIVE PANEL ERROR
            "736011" : Bool;   // (RHP_SEOC) LASER UNIT 1 READY LASER MODULE 1 IN TEST MODE
            "736012" : Bool;   // (RHP_SEOC) LASER UNIT 1 READY FAULT
            "736030" : Bool;   // (RHP_SEOC) LASER UNIT 1 ACTIVE PROGRAM NOT ACTIVE
            "736031" : Bool;   // (RHP_SEOC) LASER UNIT 1 ACTIVE NO LASER EMISSION
            "736032" : Bool;   // (RHP_SEOC) LASER UNIT 1 ACTIVE UNSAFE STATE
            "736033" : Bool;   // (RHP_SEOC) LASER UNIT 1 ACTIVE UNSAFE AREA
            "736034" : Bool;   // (RHP_SEOC) LASER UNIT 1 ACTIVE LASER-DSS ANALOG MODE MISMATCH
            "736035" : Bool;   // (RHP_SEOC) LASER UNIT 1 AXIS NOT MOVING WHILE LASER ON
            "736050" : Bool;   // (RHP_SEOC) LASER UNIT 2 READY CIRCUIT BREAKER ALARM
            "736051" : Bool;   // (RHP_SEOC) LASER UNIT 2 READY LASER ERROR
            "736052" : Bool;   // (RHP_SEOC) LASER UNIT 2 READY WARNING LASER
            "736053" : Bool;   // (RHP_SEOC) LASER UNIT 2 READY LASER NOT READY
            "736054" : Bool;   // (RHP_SEOC) LASER UNIT 2 READY LASER NOT SWITCHED ON
            "736055" : Bool;   // (RHP_SEOC) LASER UNIT 2 READY ANALOG CONTROL ERROR
            "736056" : Bool;   // (RHP_SEOC) LASER UNIT 2 READY LASER NOT ASSIGNED
            "736057" : Bool;   // (RHP_SEOC) LASER UNIT 2 READY OVERTEMPERATURE ALARM
            "736058" : Bool;   // (RHP_SEOC) LASER UNIT 2 READY LASER EMERGENCY STOP ACTIVE
            "736059" : Bool;   // (RHP_SEOC) LASER UNIT 2 READY LASER SC STATUS ACTIVE
            "736060" : Bool;   // (RHP_SEOC) LASER UNIT 2 READY ACTIVE PANEL ERROR
            "736061" : Bool;   // (RHP_SEOC) LASER UNIT 2 READY LASER MODULE 1 IN TEST MODE
            "736062" : Bool;   // (RHP_SEOC) LASER UNIT 2 READY FAULT
            "736080" : Bool;   // (RHP_SEOC) LASER UNIT 2 ACTIVE PROGRAM NOT ACTIVE
            "736081" : Bool;   // (RHP_SEOC) LASER UNIT 2 ACTIVE NO LASER EMISSION
            "736082" : Bool;   // (RHP_SEOC) LASER UNIT 2 ACTIVE UNSAFE STATE
            "736083" : Bool;   // (RHP_SEOC) LASER UNIT 2 ACTIVE UNSAFE AREA
            "736084" : Bool;   // (RHP_SEOC) LASER UNIT 2 ACTIVE LASER-DSS ANALOG MODE MISMATCH
            "736085" : Bool;   // (RHP_SEOC) LASER UNIT 2 AXIS NOT MOVING WHILE LASER ON
            "736108" : Bool;   // (RHP_SEOC) UNIT 1 LASER POINTER NOT READY ALARM
            "736109" : Bool;   // (RHP_SEOC) UNIT 2 LASER POINTER NOT READY ALARM
            "736115" : Bool;   // (IS_SEOC) UNIT 1 Z13 NOT IN FACE R CLADDING POSITION ALARM
            "736117" : Bool;   // (IS_SEOC) UNIT 2 Z23 NOT IN FACE R CLADDING POSITION ALARM
            "736220" : Bool;   // (IS_SEOC) LASER COOLING SYSTEM NOZZLE U02 FLOW LOW ALARM
            "736221" : Bool;   // (IS_SEOC) LASER COOLING SYSTEM NOZZLE U02 FLOW HIGH ALARM
            "736222" : Bool;   // (IS_SEOC) LASER COOLING SYSTEM NOZZLE U02 FLOW SETPOINT ALARM
            "736223" : Bool;   // (IS_SEOC) LASER COOLING SYSTEM NOZZLE U02 TEMPERATURE LOW ALARM
            "736224" : Bool;   // (IS_SEOC) LASER COOLING SYSTEM NOZZLE U02 TEMPERATURE HIGH ALARM
            "736225" : Bool;   // (IS_SEOC) LASER COOLING SYSTEM NOZZLE U02 TEMPERATURE SETPOINT ALARM
            "736230" : Bool;   // (IS_SEOC) LASER COOLING SYSTEM HEAD U02 FLOW LOW ALARM
            "736231" : Bool;   // (IS_SEOC) LASER COOLING SYSTEM HEAD U02 FLOW HIGH ALARM
            "736232" : Bool;   // (IS_SEOC) LASER COOLING SYSTEM HEAD U02 FLOW SETPOINT ALARM
            "736233" : Bool;   // (IS_SEOC) LASER COOLING SYSTEM HEAD U02 TEMPERATURE LOW ALARM
            "736234" : Bool;   // (IS_SEOC) LASER COOLING SYSTEM HEAD U02 TEMPERATURE HIGH ALARM
            "736235" : Bool;   // (IS_SEOC) LASER COOLING SYSTEM HEAD U02 TEMPERATURE SETPOINT ALARM
            "736240" : Bool;   // (IS_SEOC) LASER COOLING SYSTEM NOZZLE U01 FLOW LOW ALARM
            "736241" : Bool;   // (IS_SEOC) LASER COOLING SYSTEM NOZZLE U01 FLOW HIGH ALARM
            "736242" : Bool;   // (IS_SEOC) LASER COOLING SYSTEM NOZZLE U01 FLOW SETPOINT ALARM
            "736243" : Bool;   // (IS_SEOC) LASER COOLING SYSTEM NOZZLE U01 TEMPERATURE LOW ALARM
            "736244" : Bool;   // (IS_SEOC) LASER COOLING SYSTEM NOZZLE U01 TEMPERATURE HIGH ALARM
            "736245" : Bool;   // (IS_SEOC) LASER COOLING SYSTEM NOZZLE U01 TEMPERATURE SETPOINT ALARM
            "736250" : Bool;   // (IS_SEOC) LASER COOLING SYSTEM HEAD U01 FLOW LOW ALARM
            "736251" : Bool;   // (IS_SEOC) LASER COOLING SYSTEM HEAD U01 FLOW HIGH ALARM
            "736252" : Bool;   // (IS_SEOC) LASER COOLING SYSTEM HEAD U01 FLOW SETPOINT ALARM
            "736253" : Bool;   // (IS_SEOC) LASER COOLING SYSTEM HEAD U01 TEMPERATURE LOW ALARM
            "736254" : Bool;   // (IS_SEOC) LASER COOLING SYSTEM HEAD U01 TEMPERATURE HIGH ALARM
            "736255" : Bool;   // (IS_SEOC) LASER COOLING SYSTEM HEAD U01 TEMPERATURE SETPOINT ALARM
            "736260" : Bool;   // (IS_SEOC) LASER SYSTEM PROTECTION GAS U01 FLOW LOW ALARM
            "736261" : Bool;   // (IS_SEOC) LASER SYSTEM PROTECTION GAS U01 FLOW HIGH ALARM
            "736262" : Bool;   // (IS_SEOC) LASER SYSTEM PROTECTION GAS U01 TEMPERATURE LOW ALARM
            "736263" : Bool;   // (IS_SEOC) LASER SYSTEM PROTECTION GAS U01 TEMPERATURE HIGH ALARM
            "736268" : Bool;   // (IS_SEOC) LASER SYSTEM PROTECTION GAS U01 SIMULTANEITY ALARM
            "736269" : Bool;   // (IS_SEOC) LASER SYSTEM PROTECTION GAS U01 TIME EXCEEDED ALARM
            "736270" : Bool;   // (IS_SEOC) LASER SYSTEM PROTECTION GAS U01 SWITCH ON ALARM
            "736271" : Bool;   // (IS_SEOC) LASER SYSTEM PROTECTION GAS U01 SWITCH OFF ALARM
            "736278" : Bool;   // (IS_SEOC) LASER SYSTEM PROTECTION GAS U02 SIMULTANEITY ALARM
            "736279" : Bool;   // (IS_SEOC) LASER SYSTEM PROTECTION GAS U02 TIME EXCEEDED ALARM
            "736280" : Bool;   // (IS_SEOC) LASER SYSTEM PROTECTION GAS U02 SWITCH ON ALARM
            "736281" : Bool;   // (IS_SEOC) LASER SYSTEM PROTECTION GAS U02 SWITCH OFF ALARM
            "736295" : Bool;   // (IS_SEOC) LASER SYSTEM PROTECTION GAS U02 FLOW LOW ALARM
            "736296" : Bool;   // (IS_SEOC) LASER SYSTEM PROTECTION GAS U02 FLOW HIGH ALARM
            "736297" : Bool;   // (IS_SEOC) LASER SYSTEM PROTECTION GAS U02 TEMPERATURE LOW ALARM
            "736298" : Bool;   // (IS_SEOC) LASER SYSTEM PROTECTION GAS U02 TEMPERATURE HIGH ALARM
            "736310" : Bool;   // (SEOC) LASER COOLING SYSTEM OUTPUT SENSOR U01 FLOW LOW ALARM
            "736311" : Bool;   // (SEOC) LASER COOLING SYSTEM OUTPUT SENSOR U01 FLOW HIGH ALARM
            "736312" : Bool;   // (SEOC) LASER COOLING SYSTEM OUTPUT SENSOR U01 FLOW SETPOINT ALARM
            "736313" : Bool;   // (SEOC) LASER COOLING SYSTEM OUTPUT SENSOR U01 TEMPERATURE LOW ALARM
            "736314" : Bool;   // (SEOC) LASER COOLING SYSTEM OUTPUT SENSOR U01 TEMPERATURE HIGH ALARM
            "736315" : Bool;   // (SEOC) LASER COOLING SYSTEM OUTPUT SENSOR U01 TEMPERATURE SETPOINT ALARM
            "736318" : Bool;   // (SEOC) LASER COOLING SYSTEM OUTPUT SENSOR U02 FLOW LOW ALARM
            "736319" : Bool;   // (SEOC) LASER COOLING SYSTEM OUTPUT SENSOR U02 FLOW HIGH ALARM
            "736320" : Bool;   // (SEOC) LASER COOLING SYSTEM OUTPUT SENSOR U02 FLOW SETPOINT ALARM
            "736321" : Bool;   // (SEOC) LASER COOLING SYSTEM OUTPUT SENSOR U02 TEMPERATURE LOW ALARM
            "736322" : Bool;   // (SEOC) LASER COOLING SYSTEM OUTPUT SENSOR U02 TEMPERATURE HIGH ALARM
            "736323" : Bool;   // (SEOC) LASER COOLING SYSTEM OUTPUT SENSOR U02 TEMPERATURE SETPOINT ALARM
            SPARE : Struct   // SPARE ALARMS
               "736400" : Bool;   // (IS_SEOC) UNIT 1 PYROMETER PROCESS TEMPERATURE LOW ALARM
               "736401" : Bool;   // (IS_SEOC) UNIT 1 PYROMETER PROCESS TEMPERATURE HIGH ALARM
               "736402" : Bool;   // (IS_SEOC) UNIT 1 PYROMETER HEAD TEMPERATURE LOW ALARM
               "736403" : Bool;   // (IS_SEOC) UNIT 1 PYROMETER HEAD TEMPERATURE HIGH ALARM
               "736404" : Bool;   // (IS_SEOC) UNIT 1 PYROMETER EMISSIVITY LOW ALARM
               "736405" : Bool;   // (IS_SEOC) UNIT 1 PYROMETER EMISSIVITY HIGH ALARM
               "736408" : Bool;   // (IS_SEOC) UNIT 2 PYROMETER PROCESS TEMPERATURE LOW ALARM
               "736409" : Bool;   // (IS_SEOC) UNIT 2 PYROMETER PROCESS TEMPERATURE HIGH ALARM
               "736410" : Bool;   // (IS_SEOC) UNIT 2 PYROMETER HEAD TEMPERATURE LOW ALARM
               "736411" : Bool;   // (IS_SEOC) UNIT 2 PYROMETER HEAD TEMPERATURE HIGH ALARM
               "736412" : Bool;   // (IS_SEOC) UNIT 2 PYROMETER EMISSIVITY LOW ALARM
               "736413" : Bool;   // (IS_SEOC) UNIT 2 PYROMETER EMISSIVITY HIGH ALARM
               "736800" : Bool;   // (IS) UNIT 1 POWDER SYSTEM ALARM
               "736801" : Bool;   // (IS) UNIT 2 POWDER SYSTEM ALARM
               "736808" : Bool;   // (SEOC) UNIT 1 POWDER FEEDER 1 LINE 1 LOW POWDER
               "736809" : Bool;   // (SEOC) UNIT 1 POWDER FEEDER 1 LINE 2 LOW POWDER
               "736810" : Bool;   // (SEOC) UNIT 2 POWDER FEEDER 1 LINE 1 LOW POWDER
               "736811" : Bool;   // (SEOC) UNIT 2 POWDER FEEDER 1 LINE 2 LOW POWDER
               "736812" : Bool;   // (SEOC) UNIT 2 POWDER FEEDER 2 LINE 2 LOW POWDER
            END_STRUCT;
         END_STRUCT;
         WARNINGS : Struct   // WARNINGS ALARMS
            "740000" : Bool;   // (SEOC_WRN) RUN OUT CYCLE COMPLETED
            "740001" : Bool;   // (SEOC_WRN) SINGLE CYCLE COMPLETED
            "740002" : Bool;   // (WRN) RUN OUT CYCLE UNIT 1 COMPLETED
            "740003" : Bool;   // (WRN) RUN OUT CYCLE UNIT 2 COMPLETED
            "740008" : Bool;   // (SEOC_WRN) MAIN OPERATOR PANEL MANUAL MODE REQUESTED TO MODE GROUP 1
            "740009" : Bool;   // (SEOC_WRN) MAIN OPERATOR PANEL SEMIAUTO MODE REQUESTED TO MODE GROUP 1
            "740010" : Bool;   // (SEOC_WRN) MAIN OPERATOR PANEL SINGLE CYCLE MODE REQUESTED TO MODE GROUP 1
            "740011" : Bool;   // (SEOC_WRN) MAIN OPERATOR PANEL AUTOMATIC MODE REQUESTED TO MODE GROUP 1
            "740012" : Bool;   // (IS_WRN) MAIN OPERATOR PANEL STOP CYCLE REQUESTED
            "740013" : Bool;   // (RHP_WRN) MAIN OPERATOR PANEL RETURN TO HOME POSITION REQUESTED
            "740014" : Bool;   // (SEOC_WRN) MAIN OPERATOR PANEL STOP AT END OF CYCLE REQUESTED
            "740025" : Bool;   // (RHP_WRN) AUXILIARY OPERATOR PANEL RETURN TO HOME POSITION REQUESTED
            "740026" : Bool;   // (SEOC_WRN) AUXILIARY OPERATOR PANEL STOP AT END OF CYCLE REQUESTED
            "740032" : Bool;   // (SEOC_WRN) MANUAL MODE REQUESTED TO MODE GROUP 2
            "740033" : Bool;   // (SEOC_WRN) SEMIAUTO MODE REQUESTED TO MODE GROUP 2
            "740034" : Bool;   // (SEOC_WRN) SINGLE CYCLE MODE REQUESTED TO MODE GROUP 2
            "740035" : Bool;   // (SEOC_WRN) AUTOMATIC MODE REQUESTED TO MODE GROUP 2
            "740045" : Bool;   // (WRN) REMOVE HEAD PROTECTION COVER TO PERFORM GUIDEWAY CLEANING CYCLE UNIT 1
            "740046" : Bool;   // (WRN) REMOVE HEAD PROTECTION COVER TO PERFORM MAINTENANCE CYCLE UNIT 1
            "740049" : Bool;   // (WRN) REMOVE HEAD PROTECTION COVER TO PERFORM GUIDEWAY CLEANING CYCLE UNIT 2
            "740050" : Bool;   // (WRN) REMOVE HEAD PROTECTION COVER TO PERFORM MAINTENANCE CYCLE UNIT 2
            "740055" : Bool;   // (WRN) OVERRIDE 0%
            "740060" : Bool;   // (WRN) RUN-OUT UNIT 1 CYCLE SELECTED
            "740061" : Bool;   // (WRN) RUN-OUT UNIT 2 CYCLE SELECTED
            "740062" : Bool;   // (WRN) DRY CYCLE SELECTED
            "740063" : Bool;   // (WRN) SINGLE CYCLE SELECTED
            "740064" : Bool;   // (WRN) MANUAL LOADING MODE SELECTED
            "740065" : Bool;   // (WRN) MODE GROUP 1 STEP BY STEP MODE SELECTED
            "740066" : Bool;   // (WRN) MODE GROUP 1 MDA MODE SELECTED
            "740067" : Bool;   // (WRN) GANTRY ROBOT TEST SELECTED
            "740068" : Bool;   // (WRN) ROBOT DRY CYCLE SELECTED
            "740069" : Bool;   // (WRN) MODE GROUP 1 NO BA MODE SELECTED
            "740071" : Bool;   // (WRN) CALIBRATION CYCLE SELECTED
            "740072" : Bool;   // (WRN) MODE GROUP 1 CHANGE TO BA1 MODE ALARM
            "740073" : Bool;   // (WRN) MODE GROUP 1 CHANGE TO BA2 MODE ALARM
            "740074" : Bool;   // (WRN) MODE GROUP 1 CHANGE TO BA3 MODE ALARM
            "740075" : Bool;   // (WRN) MODE GROUP 1 CHANGE TO BA5 MODE ALARM
            "740077" : Bool;   // (WRN) SELECT AUTO OR SEMI MODE TO POWER ON SERVICES
            "740088" : Bool;   // (WRN) MODE GROUP 2 MDA MODE SELECTED
            "740091" : Bool;   // (WRN) MODE GROUP 2 NO BA MODE SELECTED
            "740094" : Bool;   // (WRN) MODE GROUP 2 CHANGE TO BA1 MODE ALARM
            "740095" : Bool;   // (WRN) MODE GROUP 2 CHANGE TO BA2 MODE ALARM
            "740096" : Bool;   // (WRN) MODE GROUP 2 CHANGE TO BA3 MODE ALARM
            "740097" : Bool;   // (WRN) MODE GROUP 2 CHANGE TO BA5 MODE ALARM
            "740160" : Bool;   // (WRN) POWER SUPPLY CIRCUIT BREAKER 110/120/220/230VAC TRIPPED
            "740161" : Bool;   // (WRN) ELECTRIC CABINET MACHINE LIGHTS CIRCUIT BREAKER TRIPPED
            "740162" : Bool;   // (WRN) SENTRON PAC CIRCUIT BREAKER TRIPPED
            "740163" : Bool;   // (WRN) WATTMETER CIRCUIT BREAKER TRIPPED
            "740164" : Bool;   // (WRN) ELECTRICAL CABINET DOOR OPEN
            "740165" : Bool;   // (WRN) BATTERY SITOP 85%
            "740166" : Bool;   // (WRN) LINE CONTACTOR NOT SWITCHED ON
            "740168" : Bool;   // (WRN) 0FC20 ELECTRICAL CABINET OUTLET CIRCUIT BREAKER TRIPPED ALARM
            "740169" : Bool;   // (WRN) 0FC21 ELECTRICAL CABINET OUTLET CIRCUIT BREAKER TRIPPED ALARM
            "740170" : Bool;   // (WRN) 0FC22 ELECTRICAL CABINET OUTLET CIRCUIT BREAKER TRIPPED ALARM
            "740171" : Bool;   // (WRN) 0FC23 ELECTRICAL CABINET OUTLET CIRCUIT BREAKER TRIPPED ALARM
            "740178" : Bool;   // (WRN) PROFINET INSPEKTOR PROFINET FAULT
            "740240" : Bool;   // (WRN) TEST STOP IN PROCESS
            "740241" : Bool;   // (WRN) TEST STOP COMPLETED
            "740281" : Bool;   // (WRN) SAVE ENERGY AUXILIARY SERVICES OFF
            "740282" : Bool;   // (WRN) SAVE ENERGY MAIN SERVICES OFF
            "740320" : Bool;   // (WRN) UNIT 1 MAIN SAFETY DOOR NOT CLOSED AND LOCKED
            "740321" : Bool;   // (WRN) UNIT 1 STATION 02 SAFETY DOOR NOT CLOSED AND LOCKED
            "740322" : Bool;   // (WRN) UNIT 1 STATION 04 SAFETY DOOR NOT CLOSED AND LOCKED
            "740325" : Bool;   // (WRN) UNIT 2 MAIN SAFETY DOOR NOT CLOSED AND LOCKED
            "740326" : Bool;   // (WRN) UNIT 2 STATION 02 SAFETY DOOR NOT CLOSED AND LOCKED
            "740327" : Bool;   // (WRN) UNIT 2 STATION 04 SAFETY DOOR NOT CLOSED AND LOCKED
            "740335" : Bool;   // (WRN) ROBOT SAFETY DOOR NOT CLOSED AND LOCKED
            "740336" : Bool;   // (WRN) UNIT 1 MAIN SAFETY DOOR UNLOCK WITH CYCLE RUNNING REQUESTED
            "740337" : Bool;   // (WRN) UNIT 1 STATION 02 SAFETY DOOR UNLOCK WITH CYCLE RUNNING REQUESTED
